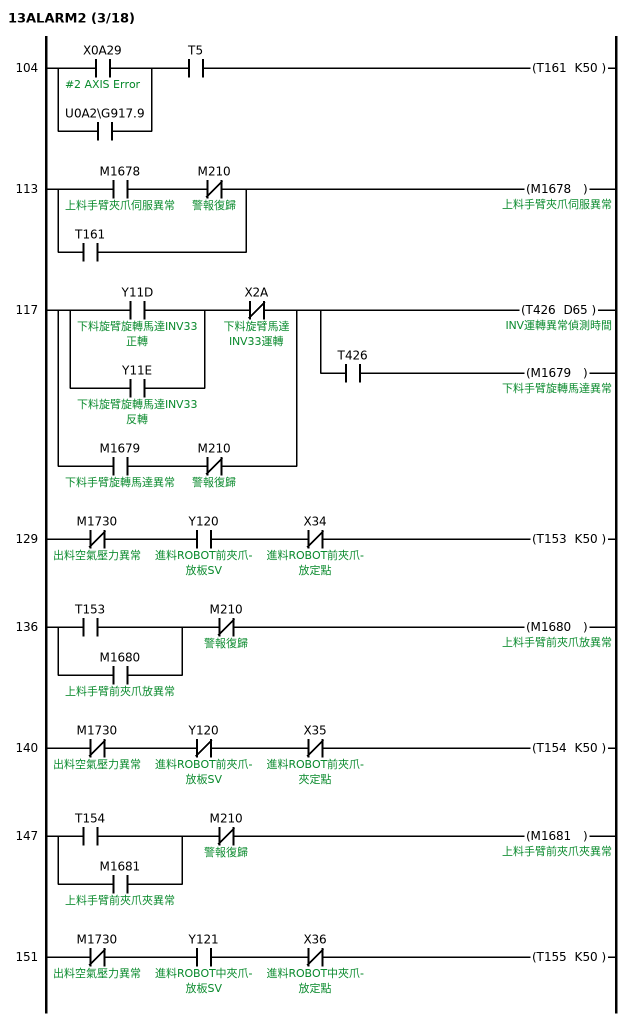
[picture p72: ladder of 13ALARM2, rungs at steps 104 to 151]
104   LD      X0A29  ; #2 AXIS Error
      OR      U0A2\G917.9
      AND     T5
      OUT     T161 K50
113   LD      M1678  ; 上料手臂夾爪伺服異常
      ANI     M210  ; 警報復歸
      OR      T161
      OUT     M1678  ; 上料手臂夾爪伺服異常
117   LD      Y11D  ; 下料旋臂旋轉馬達INV33正轉
      OR      Y11E  ; 下料旋臂旋轉馬達INV33反轉
      ANI     X2A  ; 下料旋臂馬達    INV33運轉
      LD      M1679  ; 下料手臂旋轉馬達異常
      ANI     M210  ; 警報復歸
      ORB
      OUT     T426 D65  ; INV運轉異常偵測時間
      AND     T426
      OUT     M1679  ; 下料手臂旋轉馬達異常
129   LDI     M1730  ; 出料空氣壓力異常
      AND     Y120  ; 進料ROBOT前夾爪-放板SV
      ANI     X34  ; 進料ROBOT前夾爪-放定點
      OUT     T153 K50
136   LD      T153
      OR      M1680  ; 上料手臂前夾爪放異常
      ANI     M210  ; 警報復歸
      OUT     M1680  ; 上料手臂前夾爪放異常
140   LDI     M1730  ; 出料空氣壓力異常
      ANI     Y120  ; 進料ROBOT前夾爪-放板SV
      ANI     X35  ; 進料ROBOT前夾爪-夾定點
      OUT     T154 K50
147   LD      T154
      OR      M1681  ; 上料手臂前夾爪夾異常
      ANI     M210  ; 警報復歸
      OUT     M1681  ; 上料手臂前夾爪夾異常
151   LDI     M1730  ; 出料空氣壓力異常
      AND     Y121  ; 進料ROBOT中夾爪-放板SV
      ANI     X36  ; 進料ROBOT中夾爪-放定點
      OUT     T155 K50
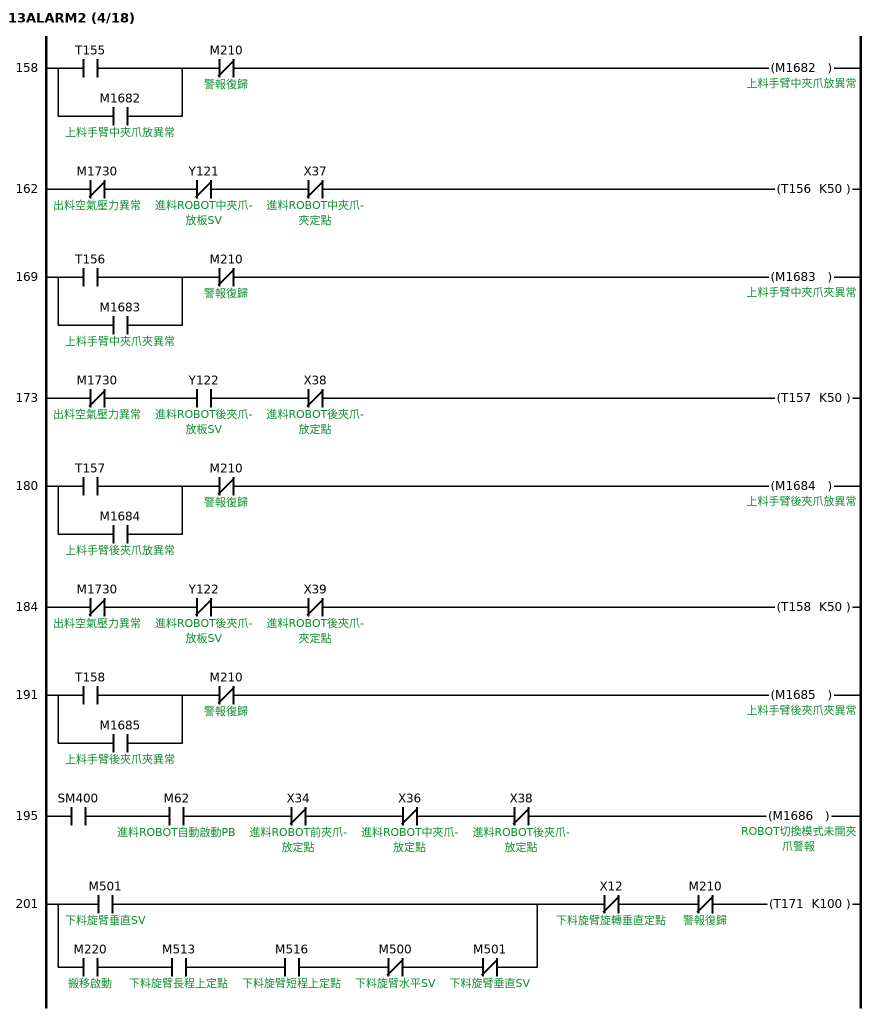
158   LD      T155
      OR      M1682  ; 上料手臂中夾爪放異常
      ANI     M210  ; 警報復歸
      OUT     M1682  ; 上料手臂中夾爪放異常
162   LDI     M1730  ; 出料空氣壓力異常
      ANI     Y121  ; 進料ROBOT中夾爪-放板SV
      ANI     X37  ; 進料ROBOT中夾爪-夾定點
      OUT     T156 K50
169   LD      T156
      OR      M1683  ; 上料手臂中夾爪夾異常
      ANI     M210  ; 警報復歸
      OUT     M1683  ; 上料手臂中夾爪夾異常
173   LDI     M1730  ; 出料空氣壓力異常
      AND     Y122  ; 進料ROBOT後夾爪-放板SV
      ANI     X38  ; 進料ROBOT後夾爪-放定點
      OUT     T157 K50
180   LD      T157
      OR      M1684  ; 上料手臂後夾爪放異常
      ANI     M210  ; 警報復歸
      OUT     M1684  ; 上料手臂後夾爪放異常
184   LDI     M1730  ; 出料空氣壓力異常
      ANI     Y122  ; 進料ROBOT後夾爪-放板SV
      ANI     X39  ; 進料ROBOT後夾爪-夾定點
      OUT     T158 K50
191   LD      T158
      OR      M1685  ; 上料手臂後夾爪夾異常
      ANI     M210  ; 警報復歸
      OUT     M1685  ; 上料手臂後夾爪夾異常
195   LD      SM400
      AND     M62  ; 進料ROBOT自動啟動PB
      ANI     X34  ; 進料ROBOT前夾爪-放定點
      ANI     X36  ; 進料ROBOT中夾爪-放定點
      ANI     X38  ; 進料ROBOT後夾爪-放定點
      OUT     M1686  ; ROBOT切換模式未開夾爪警報
201   LD      M501  ; 下料旋臂垂直SV
      LD      M220  ; 搬移啟動
      AND     M513  ; 下料旋臂長程上定點
      AND     M516  ; 下料旋臂短程上定點
      ANI     M500  ; 下料旋臂水平SV
      ANI     M501  ; 下料旋臂垂直SV
      ORB
      ANI     X12  ; 下料旋臂旋轉垂直定點
      ANI     M210  ; 警報復歸
      OUT     T171 K100
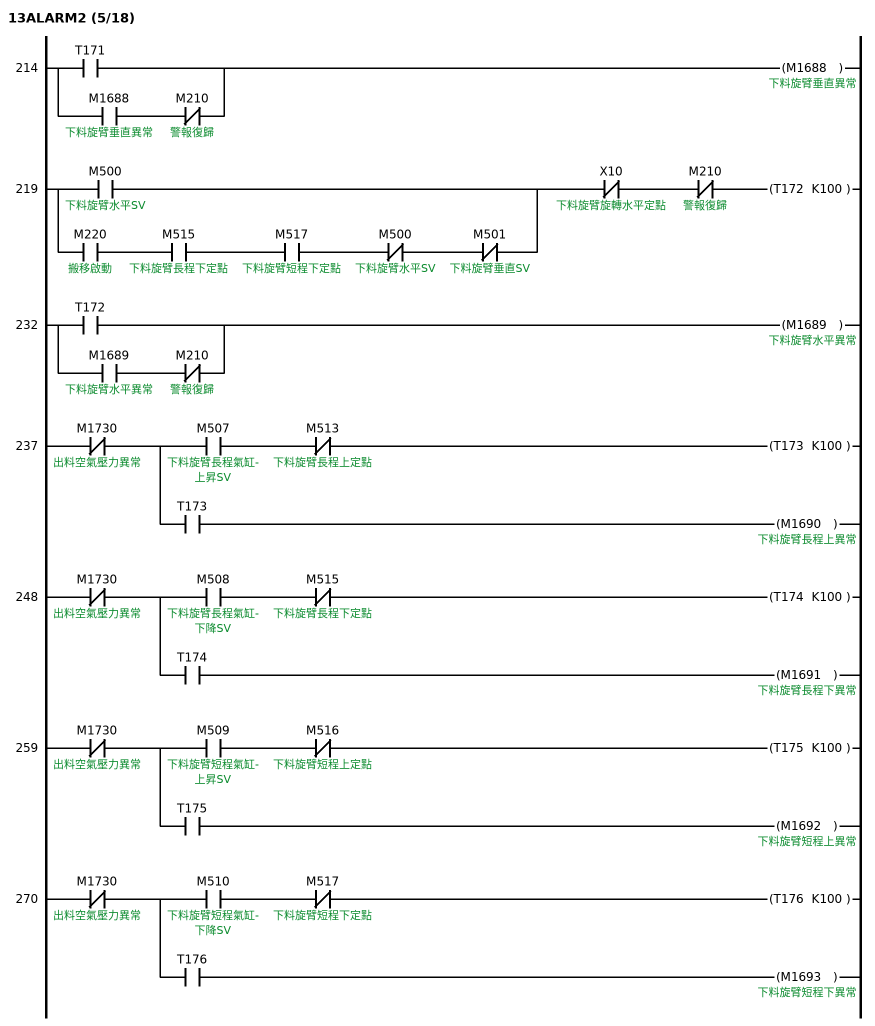
214   LD      T171
      LD      M1688  ; 下料旋臂垂直異常
      ANI     M210  ; 警報復歸
      ORB
      OUT     M1688  ; 下料旋臂垂直異常
219   LD      M500  ; 下料旋臂水平SV
      LD      M220  ; 搬移啟動
      AND     M515  ; 下料旋臂長程下定點
      AND     M517  ; 下料旋臂短程下定點
      ANI     M500  ; 下料旋臂水平SV
      ANI     M501  ; 下料旋臂垂直SV
      ORB
      ANI     X10  ; 下料旋臂旋轉水平定點
      ANI     M210  ; 警報復歸
      OUT     T172 K100
232   LD      T172
      LD      M1689  ; 下料旋臂水平異常
      ANI     M210  ; 警報復歸
      ORB
      OUT     M1689  ; 下料旋臂水平異常
237   LDI     M1730  ; 出料空氣壓力異常
      MPS
      AND     M507  ; 下料旋臂長程氣缸-上昇SV
      ANI     M513  ; 下料旋臂長程上定點
      OUT     T173 K100
      MPP
      AND     T173
      OUT     M1690  ; 下料旋臂長程上異常
248   LDI     M1730  ; 出料空氣壓力異常
      MPS
      AND     M508  ; 下料旋臂長程氣缸-下降SV
      ANI     M515  ; 下料旋臂長程下定點
      OUT     T174 K100
      MPP
      AND     T174
      OUT     M1691  ; 下料旋臂長程下異常
259   LDI     M1730  ; 出料空氣壓力異常
      MPS
      AND     M509  ; 下料旋臂短程氣缸-上昇SV
      ANI     M516  ; 下料旋臂短程上定點
      OUT     T175 K100
      MPP
      AND     T175
      OUT     M1692  ; 下料旋臂短程上異常
270   LDI     M1730  ; 出料空氣壓力異常
      MPS
      AND     M510  ; 下料旋臂短程氣缸-下降SV
      ANI     M517  ; 下料旋臂短程下定點
      OUT     T176 K100
      MPP
      AND     T176
      OUT     M1693  ; 下料旋臂短程下異常
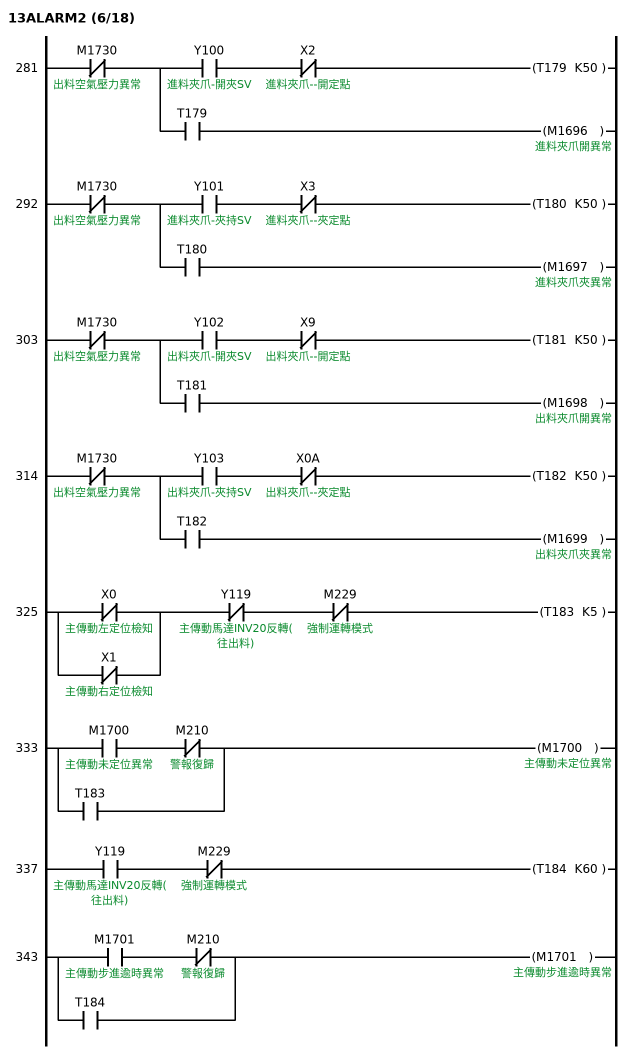
281   LDI     M1730  ; 出料空氣壓力異常
      MPS
      AND     Y100  ; 進料夾爪-開夾SV
      ANI     X2  ; 進料夾爪--開定點
      OUT     T179 K50
      MPP
      AND     T179
      OUT     M1696  ; 進料夾爪開異常
292   LDI     M1730  ; 出料空氣壓力異常
      MPS
      AND     Y101  ; 進料夾爪-夾持SV
      ANI     X3  ; 進料夾爪--夾定點
      OUT     T180 K50
      MPP
      AND     T180
      OUT     M1697  ; 進料夾爪夾異常
303   LDI     M1730  ; 出料空氣壓力異常
      MPS
      AND     Y102  ; 出料夾爪-開夾SV
      ANI     X9  ; 出料夾爪--開定點
      OUT     T181 K50
      MPP
      AND     T181
      OUT     M1698  ; 出料夾爪開異常
314   LDI     M1730  ; 出料空氣壓力異常
      MPS
      AND     Y103  ; 出料夾爪-夾持SV
      ANI     X0A  ; 出料夾爪--夾定點
      OUT     T182 K50
      MPP
      AND     T182
      OUT     M1699  ; 出料夾爪夾異常
325   LDI     X0  ; 主傳動左定位檢知
      ORI     X1  ; 主傳動右定位檢知
      ANI     Y119  ; 主傳動馬達INV20反轉(往出料)
      ANI     M229  ; 強制運轉模式
      OUT     T183 K5
333   LD      M1700  ; 主傳動未定位異常
      ANI     M210  ; 警報復歸
      OR      T183
      OUT     M1700  ; 主傳動未定位異常
337   LD      Y119  ; 主傳動馬達INV20反轉(往出料)
      ANI     M229  ; 強制運轉模式
      OUT     T184 K60
343   LD      M1701  ; 主傳動步進逾時異常
      ANI     M210  ; 警報復歸
      OR      T184
      OUT     M1701  ; 主傳動步進逾時異常
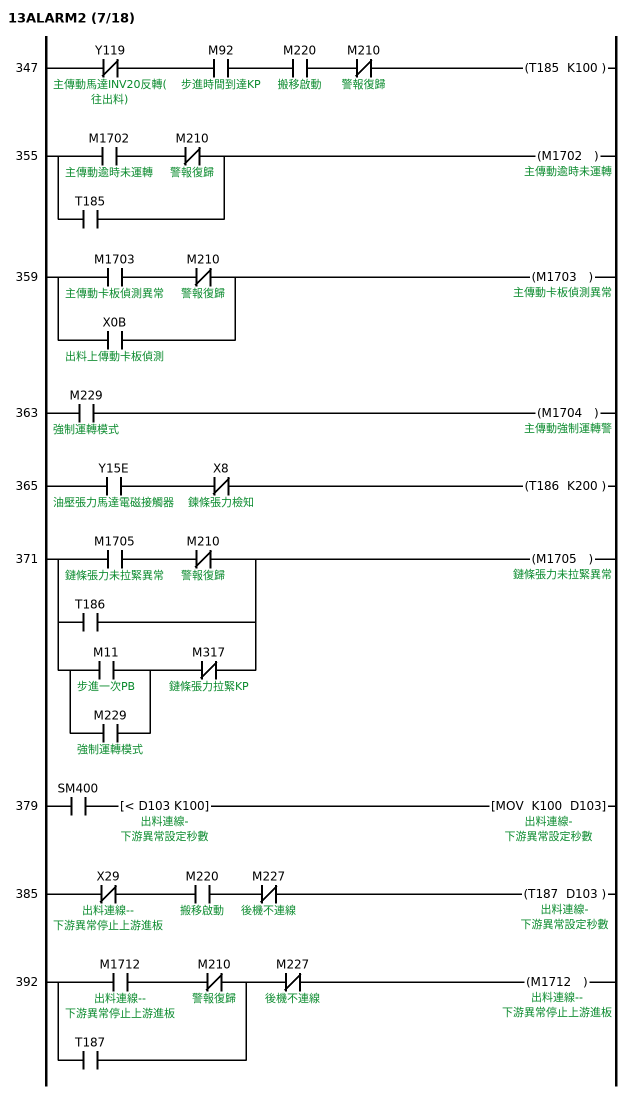
347   LDI     Y119  ; 主傳動馬達INV20反轉(往出料)
      AND     M92  ; 步進時間到達KP
      AND     M220  ; 搬移啟動
      ANI     M210  ; 警報復歸
      OUT     T185 K100
355   LD      M1702  ; 主傳動逾時未運轉
      ANI     M210  ; 警報復歸
      OR      T185
      OUT     M1702  ; 主傳動逾時未運轉
359   LD      M1703  ; 主傳動卡板偵測異常
      ANI     M210  ; 警報復歸
      OR      X0B  ; 出料上傳動卡板偵測
      OUT     M1703  ; 主傳動卡板偵測異常
363   LD      M229  ; 強制運轉模式
      OUT     M1704  ; 主傳動強制運轉警
365   LD      Y15E  ; 油壓張力馬達電磁接觸器
      ANI     X8  ; 鍊條張力檢知
      OUT     T186 K200
371   LD      M1705  ; 鏈條張力未拉緊異常
      ANI     M210  ; 警報復歸
      OR      T186
      LD      M11  ; 步進一次PB
      OR      M229  ; 強制運轉模式
      ANI     M317  ; 鏈條張力拉緊KP
      ORB
      OUT     M1705  ; 鏈條張力未拉緊異常
379   LD      SM400
      AND<    D103 K100  ; 出料連線-下游異常設定秒數
      MOV     K100 D103
385   LDI     X29  ; 出料連線--下游異常停止上游進板
      AND     M220  ; 搬移啟動
      ANI     M227  ; 後機不連線
      OUT     T187 D103  ; 出料連線-下游異常設定秒數
392   LD      M1712  ; 出料連線--下游異常停止上游進板
      ANI     M210  ; 警報復歸
      OR      T187
      ANI     M227  ; 後機不連線
      OUT     M1712  ; 出料連線--下游異常停止上游進板
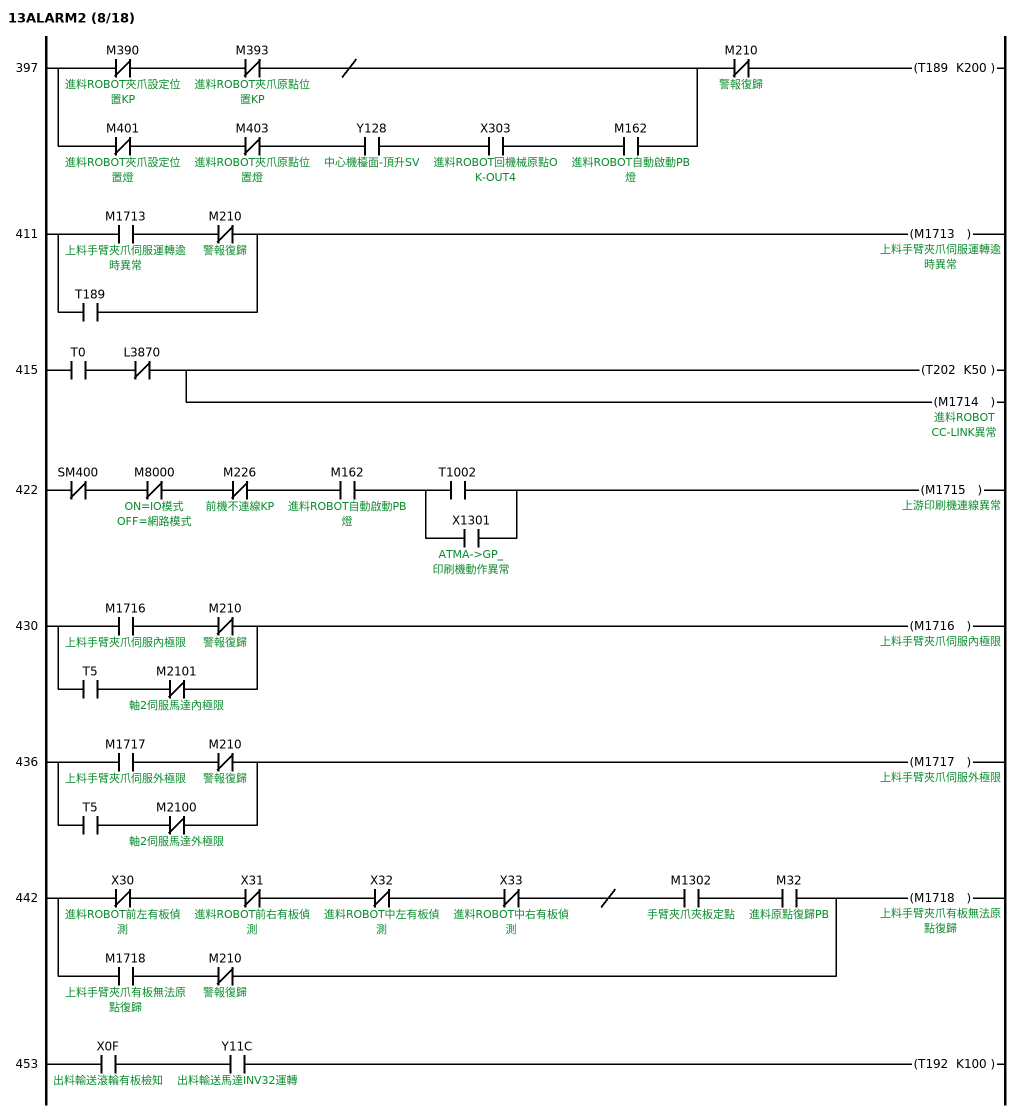
397   LDI     M390  ; 進料ROBOT夾爪設定位置KP
      ANI     M393  ; 進料ROBOT夾爪原點位置KP
      INV
      LDI     M401  ; 進料ROBOT夾爪設定位置燈
      ANI     M403  ; 進料ROBOT夾爪原點位置燈
      AND     Y128  ; 中心機檯面-頂升SV
      AND     X303  ; 進料ROBOT回機械原點OK-OUT4
      AND     M162  ; 進料ROBOT自動啟動PB燈
      ORB
      ANI     M210  ; 警報復歸
      OUT     T189 K200
411   LD      M1713  ; 上料手臂夾爪伺服運轉逾時異常
      ANI     M210  ; 警報復歸
      OR      T189
      OUT     M1713  ; 上料手臂夾爪伺服運轉逾時異常
415   LD      T0
      ANI     L3870
      OUT     T202 K50
      OUT     M1714  ; 進料ROBOT CC-LINK異常
422   LDI     SM400
      ANI     M8000  ; ON=IO模式 OFF=網路模式
      ANI     M226  ; 前機不連線KP
      AND     M162  ; 進料ROBOT自動啟動PB燈
      LD      T1002
      OR      X1301  ; ATMA->GP_印刷機動作異常
      ANB
      OUT     M1715  ; 上游印刷機連線異常
430   LD      M1716  ; 上料手臂夾爪伺服內極限
      ANI     M210  ; 警報復歸
      LD      T5
      ANI     M2101  ; 軸2伺服馬達內極限
      ORB
      OUT     M1716  ; 上料手臂夾爪伺服內極限
436   LD      M1717  ; 上料手臂夾爪伺服外極限
      ANI     M210  ; 警報復歸
      LD      T5
      ANI     M2100  ; 軸2伺服馬達外極限
      ORB
      OUT     M1717  ; 上料手臂夾爪伺服外極限
442   LDI     X30  ; 進料ROBOT前左有板偵測
      ANI     X31  ; 進料ROBOT前右有板偵測
      ANI     X32  ; 進料ROBOT中左有板偵測
      ANI     X33  ; 進料ROBOT中右有板偵測
      INV
      AND     M1302  ; 手臂夾爪夾板定點
      AND     M32  ; 進料原點復歸PB
      LD      M1718  ; 上料手臂夾爪有板無法原點復歸
      ANI     M210  ; 警報復歸
      ORB
      OUT     M1718  ; 上料手臂夾爪有板無法原點復歸
453   LD      X0F  ; 出料輸送滾輪有板檢知
      AND     Y11C  ; 出料輸送馬達INV32運轉
      OUT     T192 K100
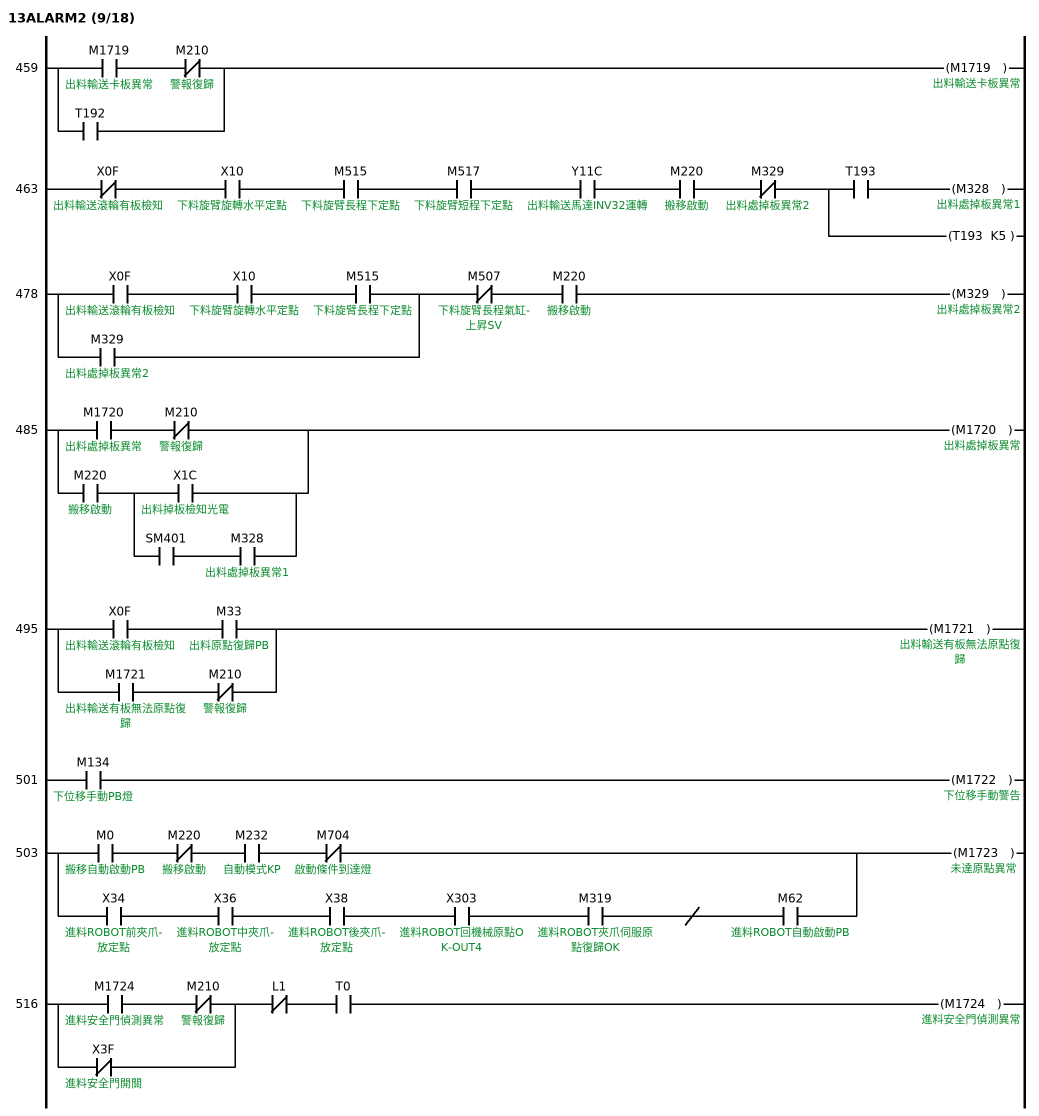
459   LD      M1719  ; 出料輸送卡板異常
      ANI     M210  ; 警報復歸
      OR      T192
      OUT     M1719  ; 出料輸送卡板異常
463   LDI     X0F  ; 出料輸送滾輪有板檢知
      AND     X10  ; 下料旋臂旋轉水平定點
      AND     M515  ; 下料旋臂長程下定點
      AND     M517  ; 下料旋臂短程下定點
      AND     Y11C  ; 出料輸送馬達INV32運轉
      AND     M220  ; 搬移啟動
      ANI     M329  ; 出料處掉板異常2
      MPS
      AND     T193
      OUT     M328  ; 出料處掉板異常1
      MPP
      OUT     T193 K5
478   LD      X0F  ; 出料輸送滾輪有板檢知
      AND     X10  ; 下料旋臂旋轉水平定點
      AND     M515  ; 下料旋臂長程下定點
      OR      M329  ; 出料處掉板異常2
      ANI     M507  ; 下料旋臂長程氣缸-上昇SV
      AND     M220  ; 搬移啟動
      OUT     M329  ; 出料處掉板異常2
485   LD      M1720  ; 出料處掉板異常
      ANI     M210  ; 警報復歸
      LD      M220  ; 搬移啟動
      LD      X1C  ; 出料掉板檢知光電
      LD      SM401
      AND     M328  ; 出料處掉板異常1
      ORB
      ANB
      ORB
      OUT     M1720  ; 出料處掉板異常
495   LD      X0F  ; 出料輸送滾輪有板檢知
      AND     M33  ; 出料原點復歸PB
      LD      M1721  ; 出料輸送有板無法原點復歸
      ANI     M210  ; 警報復歸
      ORB
      OUT     M1721  ; 出料輸送有板無法原點復歸
501   LD      M134  ; 下位移手動PB燈
      OUT     M1722  ; 下位移手動警告
503   LD      M0  ; 搬移自動啟動PB
      ANI     M220  ; 搬移啟動
      AND     M232  ; 自動模式KP
      ANI     M704  ; 啟動條件到達燈
      LD      X34  ; 進料ROBOT前夾爪-放定點
      AND     X36  ; 進料ROBOT中夾爪-放定點
      AND     X38  ; 進料ROBOT後夾爪-放定點
      AND     X303  ; 進料ROBOT回機械原點OK-OUT4
      AND     M319  ; 進料ROBOT夾爪伺服原點復歸OK
      INV
      AND     M62  ; 進料ROBOT自動啟動PB
      ORB
      OUT     M1723  ; 未達原點異常
516   LD      M1724  ; 進料安全門偵測異常
      ANI     M210  ; 警報復歸
      ORI     X3F  ; 進料安全門開關
      ANI     L1
      AND     T0
      OUT     M1724  ; 進料安全門偵測異常
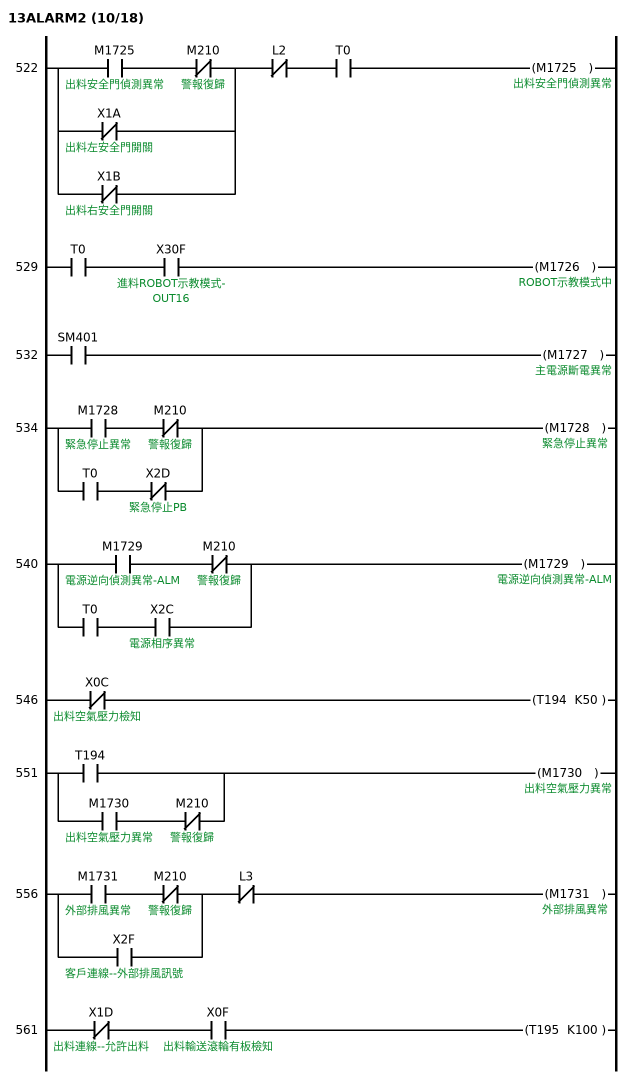
522   LD      M1725  ; 出料安全門偵測異常
      ANI     M210  ; 警報復歸
      ORI     X1A  ; 出料左安全門開關
      ORI     X1B  ; 出料右安全門開關
      ANI     L2
      AND     T0
      OUT     M1725  ; 出料安全門偵測異常
529   LD      T0
      AND     X30F  ; 進料ROBOT示教模式-OUT16
      OUT     M1726  ; ROBOT示教模式中
532   LD      SM401
      OUT     M1727  ; 主電源斷電異常
534   LD      M1728  ; 緊急停止異常
      ANI     M210  ; 警報復歸
      LD      T0
      ANI     X2D  ; 緊急停止PB
      ORB
      OUT     M1728  ; 緊急停止異常
540   LD      M1729  ; 電源逆向偵測異常-ALM
      ANI     M210  ; 警報復歸
      LD      T0
      AND     X2C  ; 電源相序異常
      ORB
      OUT     M1729  ; 電源逆向偵測異常-ALM
546   LDI     X0C  ; 出料空氣壓力檢知
      OUT     T194 K50
551   LD      T194
      LD      M1730  ; 出料空氣壓力異常
      ANI     M210  ; 警報復歸
      ORB
      OUT     M1730  ; 出料空氣壓力異常
556   LD      M1731  ; 外部排風異常
      ANI     M210  ; 警報復歸
      OR      X2F  ; 客戶連線--外部排風訊號
      ANI     L3
      OUT     M1731  ; 外部排風異常
561   LDI     X1D  ; 出料連線--允許出料
      AND     X0F  ; 出料輸送滾輪有板檢知
      OUT     T195 K100
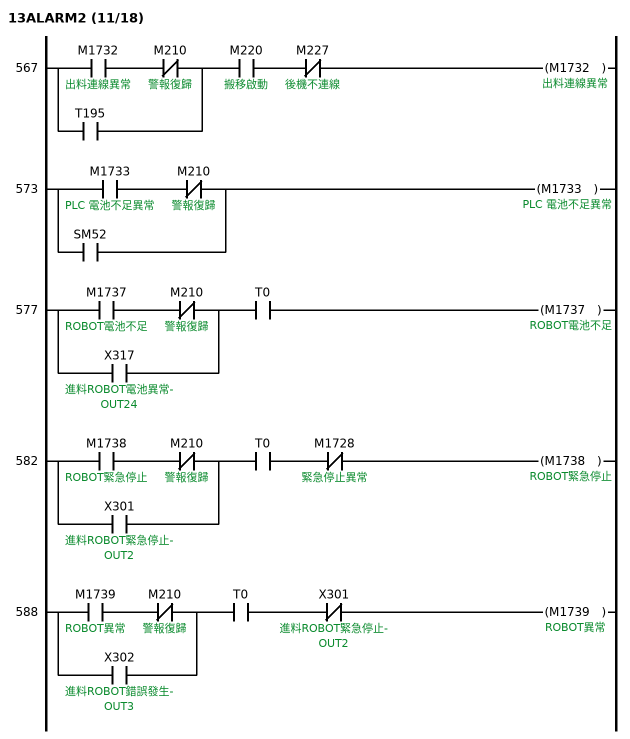
567   LD      M1732  ; 出料連線異常
      ANI     M210  ; 警報復歸
      OR      T195
      AND     M220  ; 搬移啟動
      ANI     M227  ; 後機不連線
      OUT     M1732  ; 出料連線異常
573   LD      M1733  ; PLC 電池不足異常
      ANI     M210  ; 警報復歸
      OR      SM52
      OUT     M1733  ; PLC 電池不足異常
577   LD      M1737  ; ROBOT電池不足
      ANI     M210  ; 警報復歸
      OR      X317  ; 進料ROBOT電池異常-OUT24
      AND     T0
      OUT     M1737  ; ROBOT電池不足
582   LD      M1738  ; ROBOT緊急停止
      ANI     M210  ; 警報復歸
      OR      X301  ; 進料ROBOT緊急停止-OUT2
      AND     T0
      ANI     M1728  ; 緊急停止異常
      OUT     M1738  ; ROBOT緊急停止
588   LD      M1739  ; ROBOT異常
      ANI     M210  ; 警報復歸
      OR      X302  ; 進料ROBOT錯誤發生-OUT3
      AND     T0
      ANI     X301  ; 進料ROBOT緊急停止-OUT2
      OUT     M1739  ; ROBOT異常
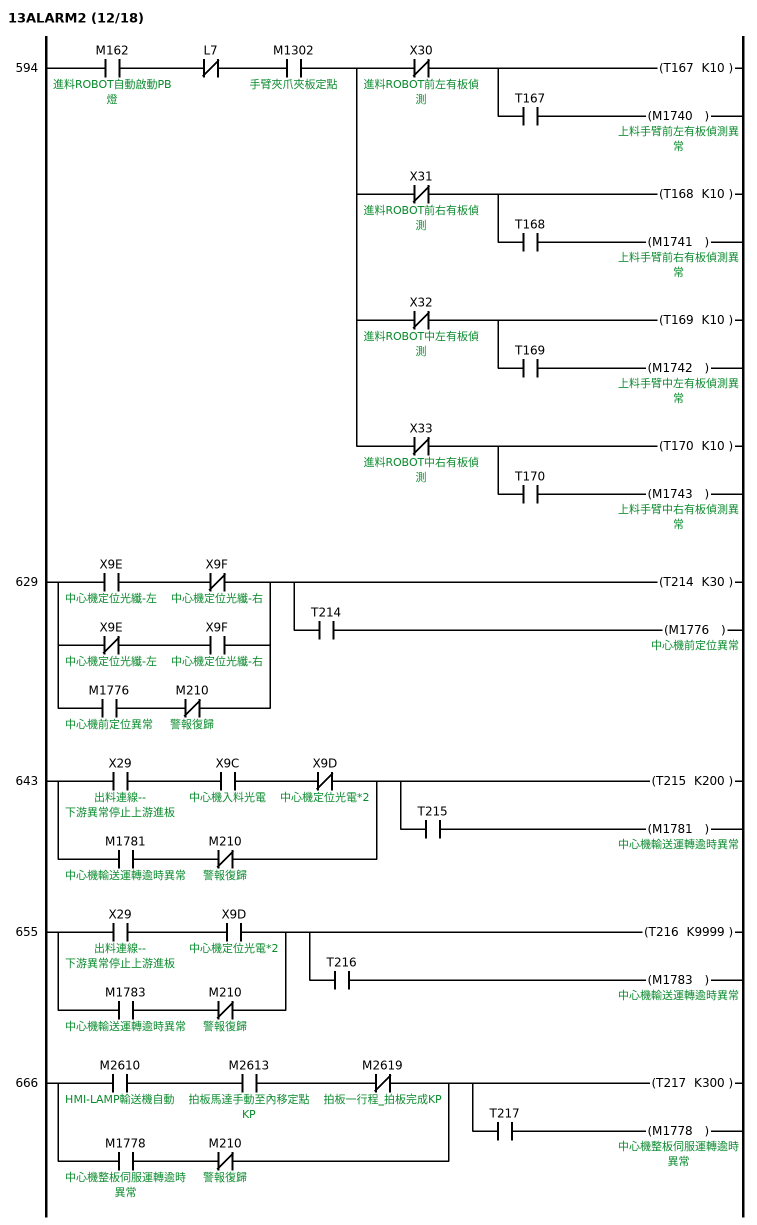
594   LD      M162  ; 進料ROBOT自動啟動PB燈
      ANI     L7
      AND     M1302  ; 手臂夾爪夾板定點
      MPS
      ANI     X30  ; 進料ROBOT前左有板偵測
      OUT     T167 K10
      AND     T167
      OUT     M1740  ; 上料手臂前左有板偵測異常
      MRD
      ANI     X31  ; 進料ROBOT前右有板偵測
      OUT     T168 K10
      AND     T168
      OUT     M1741  ; 上料手臂前右有板偵測異常
      MRD
      ANI     X32  ; 進料ROBOT中左有板偵測
      OUT     T169 K10
      AND     T169
      OUT     M1742  ; 上料手臂中左有板偵測異常
      MPP
      ANI     X33  ; 進料ROBOT中右有板偵測
      OUT     T170 K10
      AND     T170
      OUT     M1743  ; 上料手臂中右有板偵測異常
629   LD      X9E  ; 中心機定位光纖-左
      ANI     X9F  ; 中心機定位光纖-右
      LDI     X9E  ; 中心機定位光纖-左
      AND     X9F  ; 中心機定位光纖-右
      ORB
      LD      M1776  ; 中心機前定位異常
      ANI     M210  ; 警報復歸
      ORB
      OUT     T214 K30
      AND     T214
      OUT     M1776  ; 中心機前定位異常
643   LD      X29  ; 出料連線--下游異常停止上游進板
      AND     X9C  ; 中心機入料光電
      ANI     X9D  ; 中心機定位光電*2
      LD      M1781  ; 中心機輸送運轉逾時異常
      ANI     M210  ; 警報復歸
      ORB
      OUT     T215 K200
      AND     T215
      OUT     M1781  ; 中心機輸送運轉逾時異常
655   LD      X29  ; 出料連線--下游異常停止上游進板
      AND     X9D  ; 中心機定位光電*2
      LD      M1783  ; 中心機輸送運轉逾時異常
      ANI     M210  ; 警報復歸
      ORB
      OUT     T216 K9999
      AND     T216
      OUT     M1783  ; 中心機輸送運轉逾時異常
666   LD      M2610  ; HMI-LAMP輸送機自動
      AND     M2613  ; 拍板馬達手動至內移定點KP
      ANI     M2619  ; 拍板一行程_拍板完成KP
      LD      M1778  ; 中心機整板伺服運轉逾時異常
      ANI     M210  ; 警報復歸
      ORB
      OUT     T217 K300
      AND     T217
      OUT     M1778  ; 中心機整板伺服運轉逾時異常
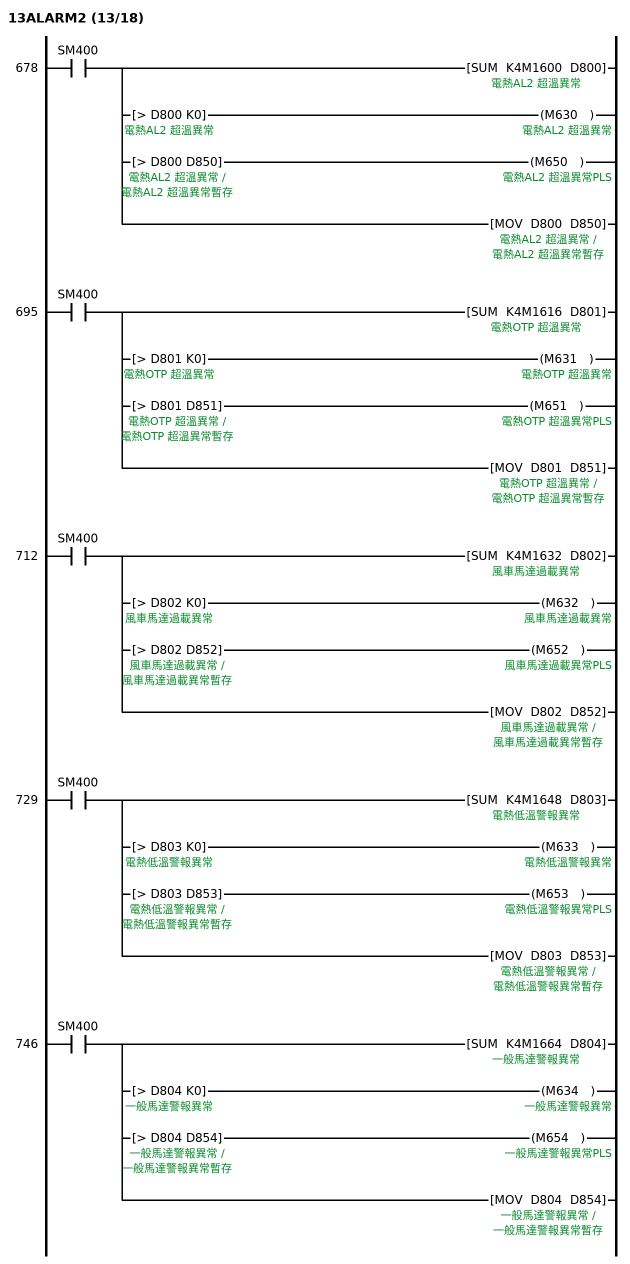
678   LD      SM400
      SUM     K4M1600 D800  ; #01 電熱AL2 超溫 / 電熱AL2 超溫異常
      MPS
      AND>    D800 K0  ; 電熱AL2 超溫異常
      OUT     M630  ; 電熱AL2 超溫異常
      MRD
      AND>    D800 D850  ; 電熱AL2 超溫異常 / 電熱AL2 超溫異常暫存
      OUT     M650  ; 電熱AL2 超溫異常PLS
      MPP
      MOV     D800 D850
695   LD      SM400
      SUM     K4M1616 D801  ; #01 電熱OTP 超溫 / 電熱OTP 超溫異常
      MPS
      AND>    D801 K0  ; 電熱OTP 超溫異常
      OUT     M631  ; 電熱OTP 超溫異常
      MRD
      AND>    D801 D851  ; 電熱OTP 超溫異常 / 電熱OTP 超溫異常暫存
      OUT     M651  ; 電熱OTP 超溫異常PLS
      MPP
      MOV     D801 D851
712   LD      SM400
      SUM     K4M1632 D802  ; #01 風車過載 / 風車馬達過載異常
      MPS
      AND>    D802 K0  ; 風車馬達過載異常
      OUT     M632  ; 風車馬達過載異常
      MRD
      AND>    D802 D852  ; 風車馬達過載異常 / 風車馬達過載異常暫存
      OUT     M652  ; 風車馬達過載異常PLS
      MPP
      MOV     D802 D852
729   LD      SM400
      SUM     K4M1648 D803  ; #01 低溫警報 / 電熱低溫警報異常
      MPS
      AND>    D803 K0  ; 電熱低溫警報異常
      OUT     M633  ; 電熱低溫警報異常
      MRD
      AND>    D803 D853  ; 電熱低溫警報異常 / 電熱低溫警報異常暫存
      OUT     M653  ; 電熱低溫警報異常PLS
      MPP
      MOV     D803 D853
746   LD      SM400
      SUM     K4M1664 D804  ; 一般馬達警報異常
      MPS
      AND>    D804 K0  ; 一般馬達警報異常
      OUT     M634  ; 一般馬達警報異常
      MRD
      AND>    D804 D854  ; 一般馬達警報異常 / 一般馬達警報異常暫存
      OUT     M654  ; 一般馬達警報異常PLS
      MPP
      MOV     D804 D854
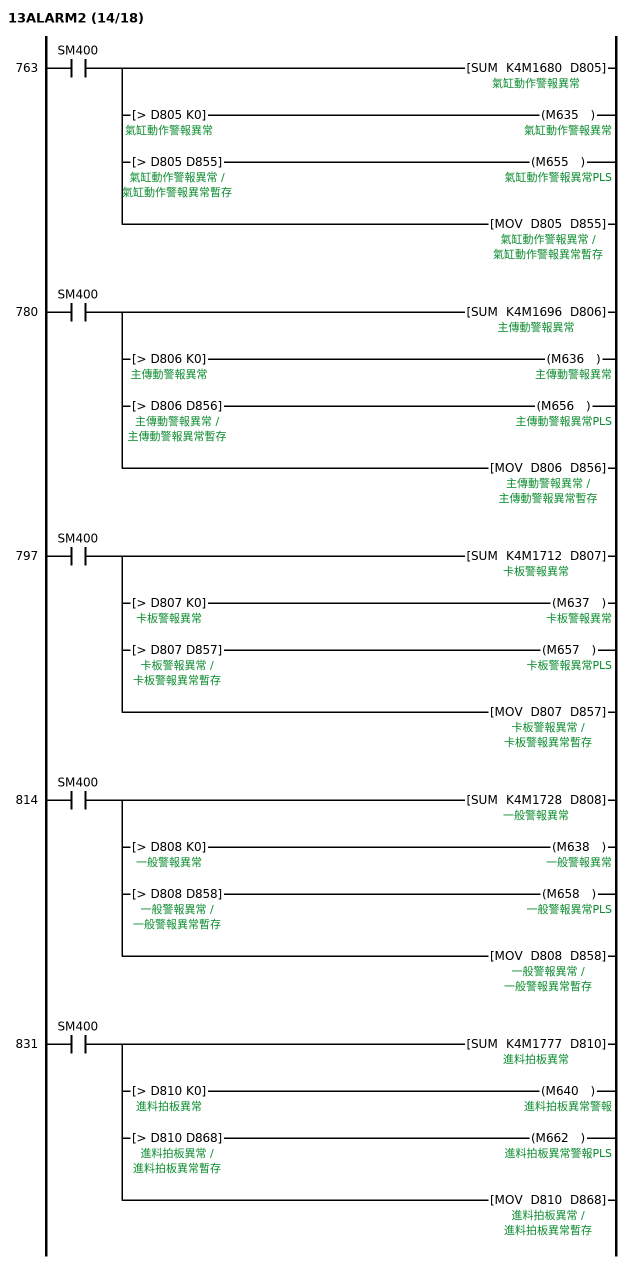
763   LD      SM400
      SUM     K4M1680 D805  ; 氣缸動作警報異常
      MPS
      AND>    D805 K0  ; 氣缸動作警報異常
      OUT     M635  ; 氣缸動作警報異常
      MRD
      AND>    D805 D855  ; 氣缸動作警報異常 / 氣缸動作警報異常暫存
      OUT     M655  ; 氣缸動作警報異常PLS
      MPP
      MOV     D805 D855
780   LD      SM400
      SUM     K4M1696 D806  ; 主傳動警報異常
      MPS
      AND>    D806 K0  ; 主傳動警報異常
      OUT     M636  ; 主傳動警報異常
      MRD
      AND>    D806 D856  ; 主傳動警報異常 / 主傳動警報異常暫存
      OUT     M656  ; 主傳動警報異常PLS
      MPP
      MOV     D806 D856
797   LD      SM400
      SUM     K4M1712 D807  ; 卡板警報異常
      MPS
      AND>    D807 K0  ; 卡板警報異常
      OUT     M637  ; 卡板警報異常
      MRD
      AND>    D807 D857  ; 卡板警報異常 / 卡板警報異常暫存
      OUT     M657  ; 卡板警報異常PLS
      MPP
      MOV     D807 D857
814   LD      SM400
      SUM     K4M1728 D808  ; 一般警報異常
      MPS
      AND>    D808 K0  ; 一般警報異常
      OUT     M638  ; 一般警報異常
      MRD
      AND>    D808 D858  ; 一般警報異常 / 一般警報異常暫存
      OUT     M658  ; 一般警報異常PLS
      MPP
      MOV     D808 D858
831   LD      SM400
      SUM     K4M1777 D810  ; 輸送機輸送變頻器異常-ALM / 進料拍板異常
      MPS
      AND>    D810 K0  ; 進料拍板異常
      OUT     M640  ; 進料拍板異常警報
      MRD
      AND>    D810 D868  ; 進料拍板異常 / 進料拍板異常暫存
      OUT     M662  ; 進料拍板異常警報PLS
      MPP
      MOV     D810 D868
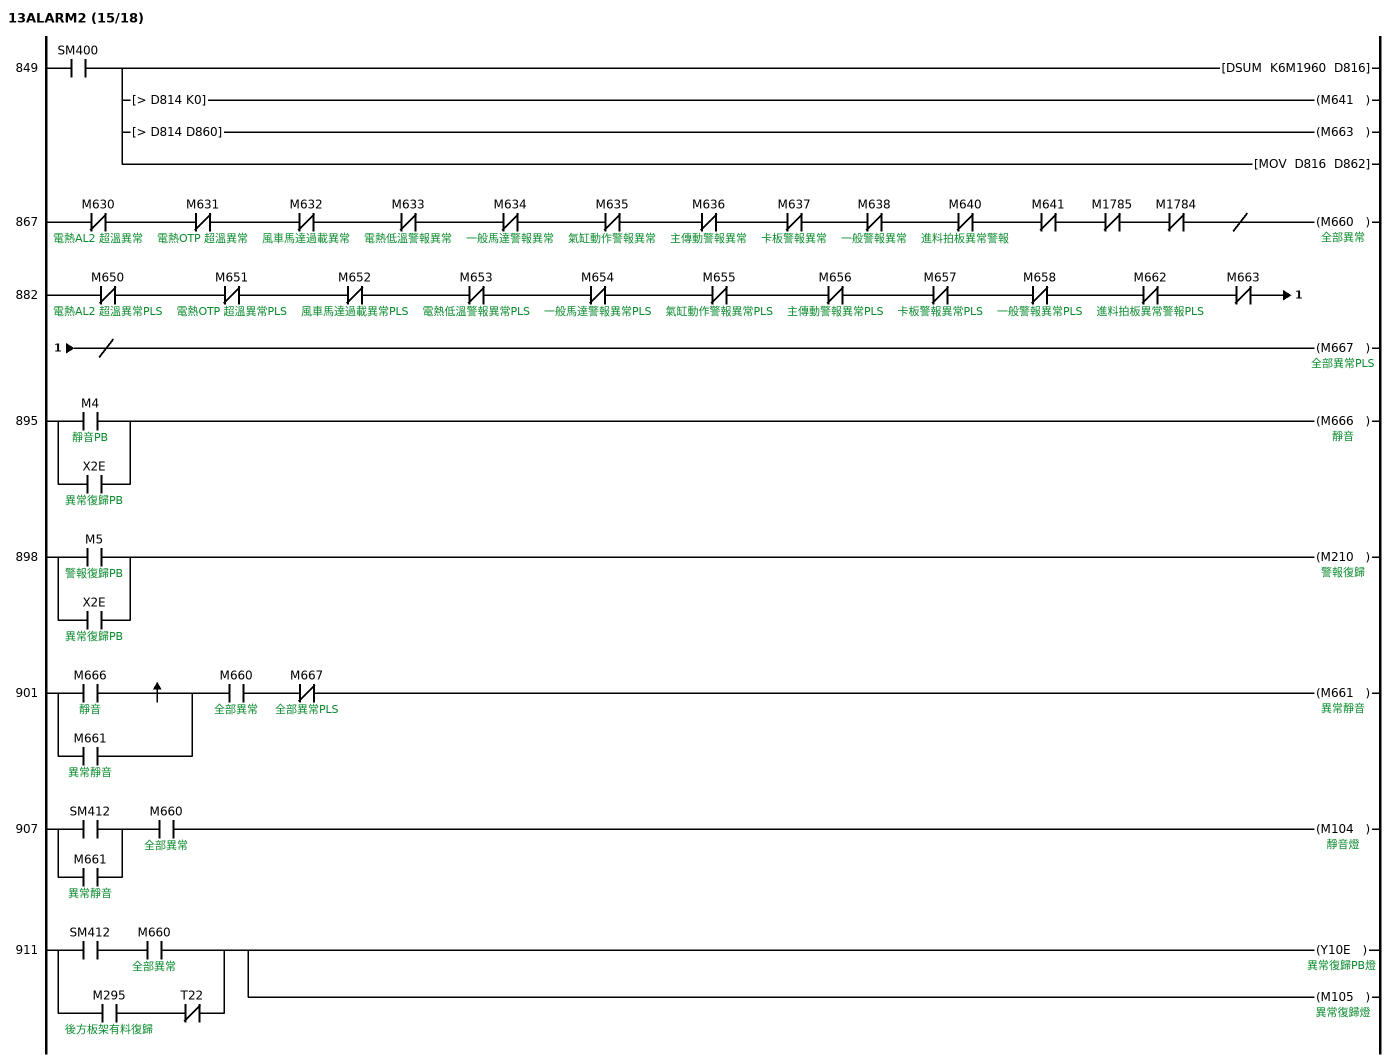
849   LD      SM400
      DSUM    K6M1960 D816
      MPS
      AND>    D814 K0
      OUT     M641
      MRD
      AND>    D814 D860
      OUT     M663
      MPP
      MOV     D816 D862
867   LDI     M630  ; 電熱AL2 超溫異常
      ANI     M631  ; 電熱OTP 超溫異常
      ANI     M632  ; 風車馬達過載異常
      ANI     M633  ; 電熱低溫警報異常
      ANI     M634  ; 一般馬達警報異常
      ANI     M635  ; 氣缸動作警報異常
      ANI     M636  ; 主傳動警報異常
      ANI     M637  ; 卡板警報異常
      ANI     M638  ; 一般警報異常
      ANI     M640  ; 進料拍板異常警報
      ANI     M641
      ANI     M1785
      ANI     M1784
      INV
      OUT     M660  ; 全部異常
882   LDI     M650  ; 電熱AL2 超溫異常PLS
      ANI     M651  ; 電熱OTP 超溫異常PLS
      ANI     M652  ; 風車馬達過載異常PLS
      ANI     M653  ; 電熱低溫警報異常PLS
      ANI     M654  ; 一般馬達警報異常PLS
      ANI     M655  ; 氣缸動作警報異常PLS
      ANI     M656  ; 主傳動警報異常PLS
      ANI     M657  ; 卡板警報異常PLS
      ANI     M658  ; 一般警報異常PLS
      ANI     M662  ; 進料拍板異常警報PLS
      ANI     M663
      INV
      OUT     M667  ; 全部異常PLS
895   LD      M4  ; 靜音PB
      OR      X2E  ; 異常復歸PB
      OUT     M666  ; 靜音
898   LD      M5  ; 警報復歸PB
      OR      X2E  ; 異常復歸PB
      OUT     M210  ; 警報復歸
901   LD      M666  ; 靜音
      MEP
      OR      M661  ; 異常靜音
      AND     M660  ; 全部異常
      ANI     M667  ; 全部異常PLS
      OUT     M661  ; 異常靜音
907   LD      SM412
      OR      M661  ; 異常靜音
      AND     M660  ; 全部異常
      OUT     M104  ; 靜音燈
911   LD      SM412
      AND     M660  ; 全部異常
      LD      M295  ; 後方板架有料復歸
      ANI     T22
      ORB
      OUT     Y10E  ; 異常復歸PB燈
      OUT     M105  ; 異常復歸燈
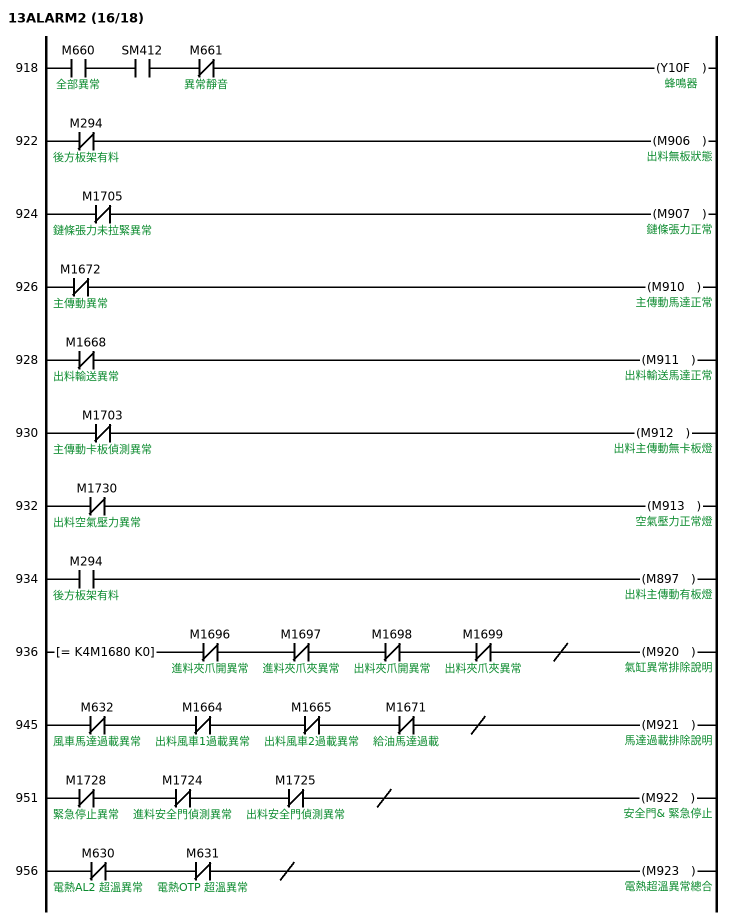
918   LD      M660  ; 全部異常
      AND     SM412
      ANI     M661  ; 異常靜音
      OUT     Y10F  ; 蜂鳴器
922   LDI     M294  ; 後方板架有料
      OUT     M906  ; 出料無板狀態
924   LDI     M1705  ; 鏈條張力未拉緊異常
      OUT     M907  ; 鏈條張力正常
926   LDI     M1672  ; 主傳動異常
      OUT     M910  ; 主傳動馬達正常
928   LDI     M1668  ; 出料輸送異常
      OUT     M911  ; 出料輸送馬達正常
930   LDI     M1703  ; 主傳動卡板偵測異常
      OUT     M912  ; 出料主傳動無卡板燈
932   LDI     M1730  ; 出料空氣壓力異常
      OUT     M913  ; 空氣壓力正常燈
934   LD      M294  ; 後方板架有料
      OUT     M897  ; 出料主傳動有板燈
936   LD=     K4M1680 K0  ; 上料手臂前夾爪放異常
      ANI     M1696  ; 進料夾爪開異常
      ANI     M1697  ; 進料夾爪夾異常
      ANI     M1698  ; 出料夾爪開異常
      ANI     M1699  ; 出料夾爪夾異常
      INV
      OUT     M920  ; 氣缸異常排除說明
945   LDI     M632  ; 風車馬達過載異常
      ANI     M1664  ; 出料風車1過載異常
      ANI     M1665  ; 出料風車2過載異常
      ANI     M1671  ; 給油馬達過載
      INV
      OUT     M921  ; 馬達過載排除說明
951   LDI     M1728  ; 緊急停止異常
      ANI     M1724  ; 進料安全門偵測異常
      ANI     M1725  ; 出料安全門偵測異常
      INV
      OUT     M922  ; 安全門& 緊急停止
956   LDI     M630  ; 電熱AL2 超溫異常
      ANI     M631  ; 電熱OTP 超溫異常
      INV
      OUT     M923  ; 電熱超溫異常總合
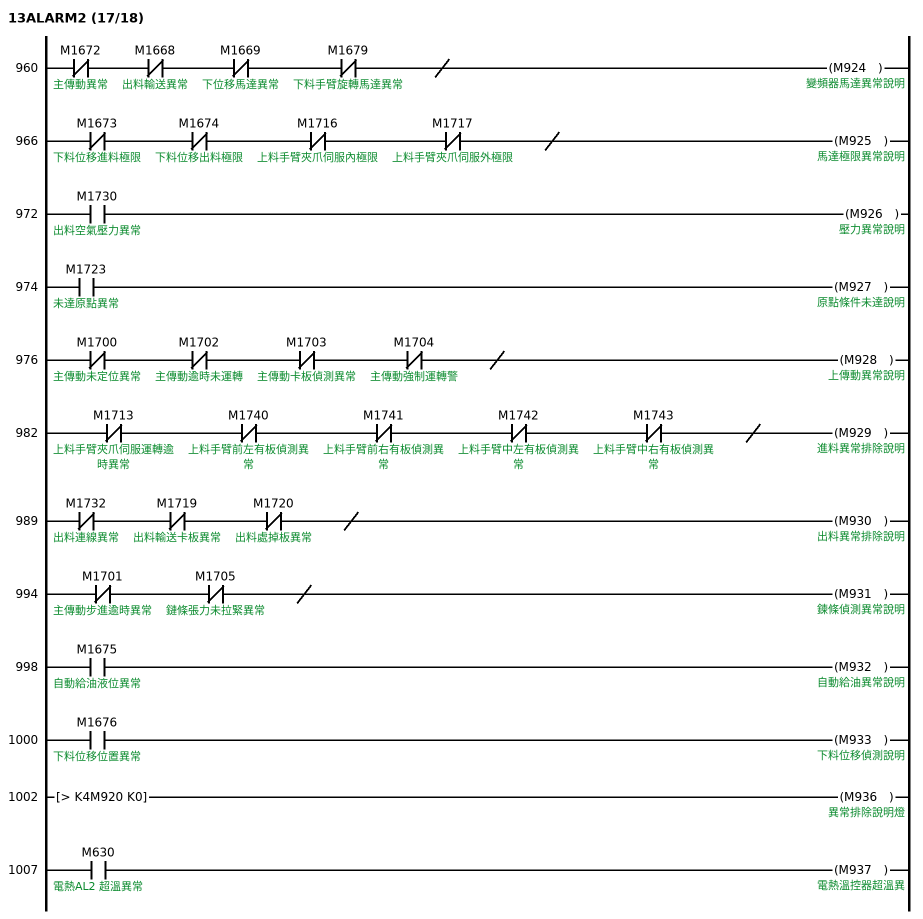
960   LDI     M1672  ; 主傳動異常
      ANI     M1668  ; 出料輸送異常
      ANI     M1669  ; 下位移馬達異常
      ANI     M1679  ; 下料手臂旋轉馬達異常
      INV
      OUT     M924  ; 變頻器馬達異常說明
966   LDI     M1673  ; 下料位移進料極限
      ANI     M1674  ; 下料位移出料極限
      ANI     M1716  ; 上料手臂夾爪伺服內極限
      ANI     M1717  ; 上料手臂夾爪伺服外極限
      INV
      OUT     M925  ; 馬達極限異常說明
972   LD      M1730  ; 出料空氣壓力異常
      OUT     M926  ; 壓力異常說明
974   LD      M1723  ; 未達原點異常
      OUT     M927  ; 原點條件未達說明
976   LDI     M1700  ; 主傳動未定位異常
      ANI     M1702  ; 主傳動逾時未運轉
      ANI     M1703  ; 主傳動卡板偵測異常
      ANI     M1704  ; 主傳動強制運轉警
      INV
      OUT     M928  ; 上傳動異常說明
982   LDI     M1713  ; 上料手臂夾爪伺服運轉逾時異常
      ANI     M1740  ; 上料手臂前左有板偵測異常
      ANI     M1741  ; 上料手臂前右有板偵測異常
      ANI     M1742  ; 上料手臂中左有板偵測異常
      ANI     M1743  ; 上料手臂中右有板偵測異常
      INV
      OUT     M929  ; 進料異常排除說明
989   LDI     M1732  ; 出料連線異常
      ANI     M1719  ; 出料輸送卡板異常
      ANI     M1720  ; 出料處掉板異常
      INV
      OUT     M930  ; 出料異常排除說明
994   LDI     M1701  ; 主傳動步進逾時異常
      ANI     M1705  ; 鏈條張力未拉緊異常
      INV
      OUT     M931  ; 鍊條偵測異常說明
998   LD      M1675  ; 自動給油液位異常
      OUT     M932  ; 自動給油異常說明
1000  LD      M1676  ; 下料位移位置異常
      OUT     M933  ; 下料位移偵測說明
1002  LD>     K4M920 K0  ; 氣缸異常排除說明
      OUT     M936  ; 異常排除說明燈
1007  LD      M630  ; 電熱AL2 超溫異常
      OUT     M937  ; 電熱溫控器超溫異
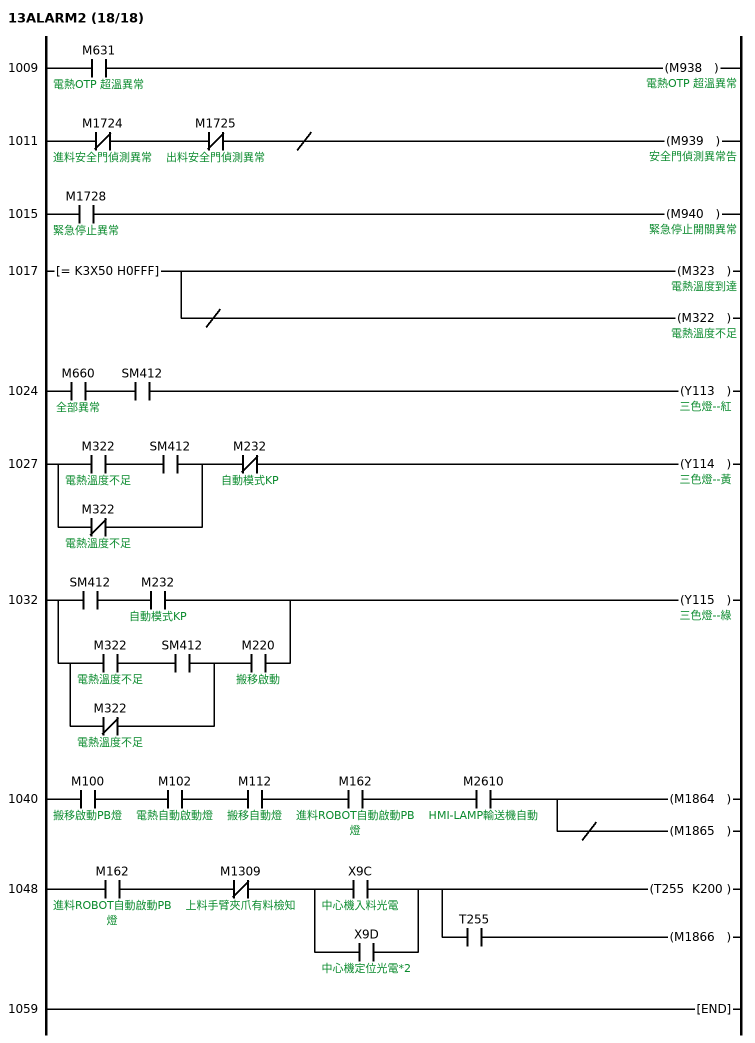
1009  LD      M631  ; 電熱OTP 超溫異常
      OUT     M938  ; 電熱OTP 超溫異常
1011  LDI     M1724  ; 進料安全門偵測異常
      ANI     M1725  ; 出料安全門偵測異常
      INV
      OUT     M939  ; 安全門偵測異常告
1015  LD      M1728  ; 緊急停止異常
      OUT     M940  ; 緊急停止開關異常
1017  LD=     K3X50 H0FFF  ; NO,01   溫度到達AL1
      OUT     M323  ; 電熱溫度到達
      INV
      OUT     M322  ; 電熱溫度不足
1024  LD      M660  ; 全部異常
      AND     SM412
      OUT     Y113  ; 三色燈--紅
1027  LD      M322  ; 電熱溫度不足
      AND     SM412
      ORI     M322  ; 電熱溫度不足
      ANI     M232  ; 自動模式KP
      OUT     Y114  ; 三色燈--黃
1032  LD      SM412
      AND     M232  ; 自動模式KP
      LD      M322  ; 電熱溫度不足
      AND     SM412
      ORI     M322  ; 電熱溫度不足
      AND     M220  ; 搬移啟動
      ORB
      OUT     Y115  ; 三色燈--綠
1040  LD      M100  ; 搬移啟動PB燈
      AND     M102  ; 電熱自動啟動燈
      AND     M112  ; 搬移自動燈
      AND     M162  ; 進料ROBOT自動啟動PB燈
      AND     M2610  ; HMI-LAMP輸送機自動
      OUT     M1864
      INV
      OUT     M1865
1048  LD      M162  ; 進料ROBOT自動啟動PB燈
      ANI     M1309  ; 上料手臂夾爪有料檢知
      LD      X9C  ; 中心機入料光電
      OR      X9D  ; 中心機定位光電*2
      ANB
      OUT     T255 K200
      AND     T255
      OUT     M1866
1059  END
END_PROGRAM

PROGRAM 14TIME
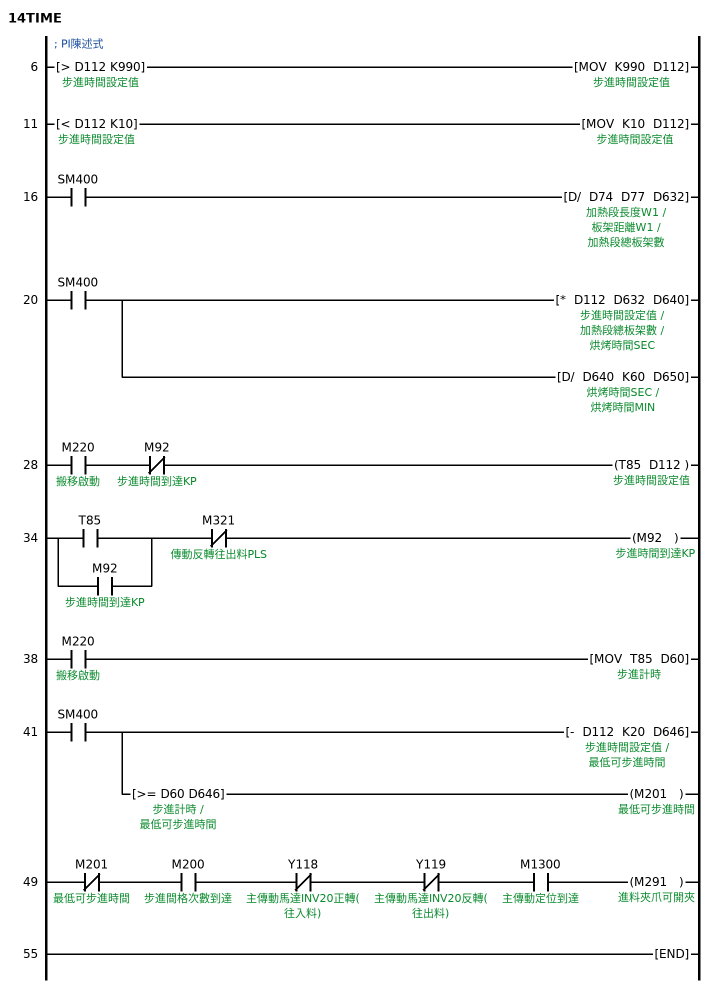
; PI陳述式
6     LD>     D112 K990  ; 步進時間設定值
      MOV     K990 D112
11    LD<     D112 K10  ; 步進時間設定值
      MOV     K10 D112
16    LD      SM400
      D/      D74 D77 D632  ; 加熱段長度W1 / 板架距離W1 / 加熱段總板架數
20    LD      SM400
      *       D112 D632 D640  ; 烘烤時間SEC
      D/      D640 K60 D650  ; 烘烤時間MIN
28    LD      M220  ; 搬移啟動
      ANI     M92  ; 步進時間到達KP
      OUT     T85 D112  ; 步進時間設定值
34    LD      T85
      OR      M92  ; 步進時間到達KP
      ANI     M321  ; 傳動反轉往出料PLS
      OUT     M92  ; 步進時間到達KP
38    LD      M220  ; 搬移啟動
      MOV     T85 D60  ; 步進計時
41    LD      SM400
      -       D112 K20 D646  ; 最低可步進時間
      AND>=   D60 D646  ; 步進計時 / 最低可步進時間
      OUT     M201  ; 最低可步進時間
49    LDI     M201  ; 最低可步進時間
      AND     M200  ; 步進間格次數到達
      ANI     Y118  ; 主傳動馬達INV20正轉(往入料)
      ANI     Y119  ; 主傳動馬達INV20反轉(往出料)
      AND     M1300  ; 主傳動定位到達
      OUT     M291  ; 進料夾爪可開夾
55    END
END_PROGRAM

PROGRAM 15STATUS
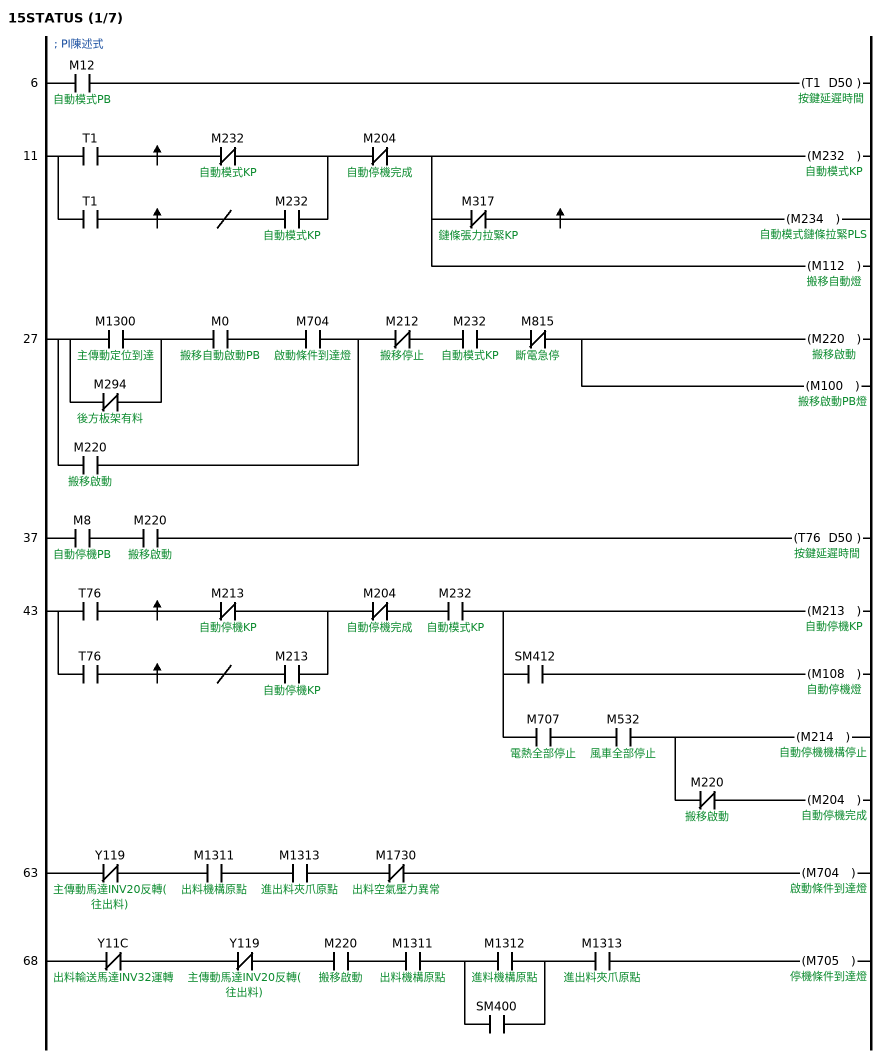
; PI陳述式
6     LD      M12  ; 自動模式PB
      OUT     T1 D50  ; 按鍵延遲時間
11    LD      T1
      MEP
      ANI     M232  ; 自動模式KP
      LD      T1
      MEP
      INV
      AND     M232  ; 自動模式KP
      ORB
      ANI     M204  ; 自動停機完成
      OUT     M232  ; 自動模式KP
      MPS
      ANI     M317  ; 鏈條張力拉緊KP
      MEP
      OUT     M234  ; 自動模式鏈條拉緊PLS
      MPP
      OUT     M112  ; 搬移自動燈
27    LD      M1300  ; 主傳動定位到達
      ORI     M294  ; 後方板架有料
      AND     M0  ; 搬移自動啟動PB
      AND     M704  ; 啟動條件到達燈
      OR      M220  ; 搬移啟動
      ANI     M212  ; 搬移停止
      AND     M232  ; 自動模式KP
      ANI     M815  ; 斷電急停
      OUT     M220  ; 搬移啟動
      OUT     M100  ; 搬移啟動PB燈
37    LD      M8  ; 自動停機PB
      AND     M220  ; 搬移啟動
      OUT     T76 D50  ; 按鍵延遲時間
43    LD      T76
      MEP
      ANI     M213  ; 自動停機KP
      LD      T76
      MEP
      INV
      AND     M213  ; 自動停機KP
      ORB
      ANI     M204  ; 自動停機完成
      AND     M232  ; 自動模式KP
      OUT     M213  ; 自動停機KP
      MPS
      AND     SM412
      OUT     M108  ; 自動停機燈
      MPP
      AND     M707  ; 電熱全部停止
      AND     M532  ; 風車全部停止
      OUT     M214  ; 自動停機機構停止
      ANI     M220  ; 搬移啟動
      OUT     M204  ; 自動停機完成
63    LDI     Y119  ; 主傳動馬達INV20反轉(往出料)
      AND     M1311  ; 出料機構原點
      AND     M1313  ; 進出料夾爪原點
      ANI     M1730  ; 出料空氣壓力異常
      OUT     M704  ; 啟動條件到達燈
68    LDI     Y11C  ; 出料輸送馬達INV32運轉
      ANI     Y119  ; 主傳動馬達INV20反轉(往出料)
      AND     M220  ; 搬移啟動
      AND     M1311  ; 出料機構原點
      LD      M1312  ; 進料機構原點
      OR      SM400
      ANB
      AND     M1313  ; 進出料夾爪原點
      OUT     M705  ; 停機條件到達燈
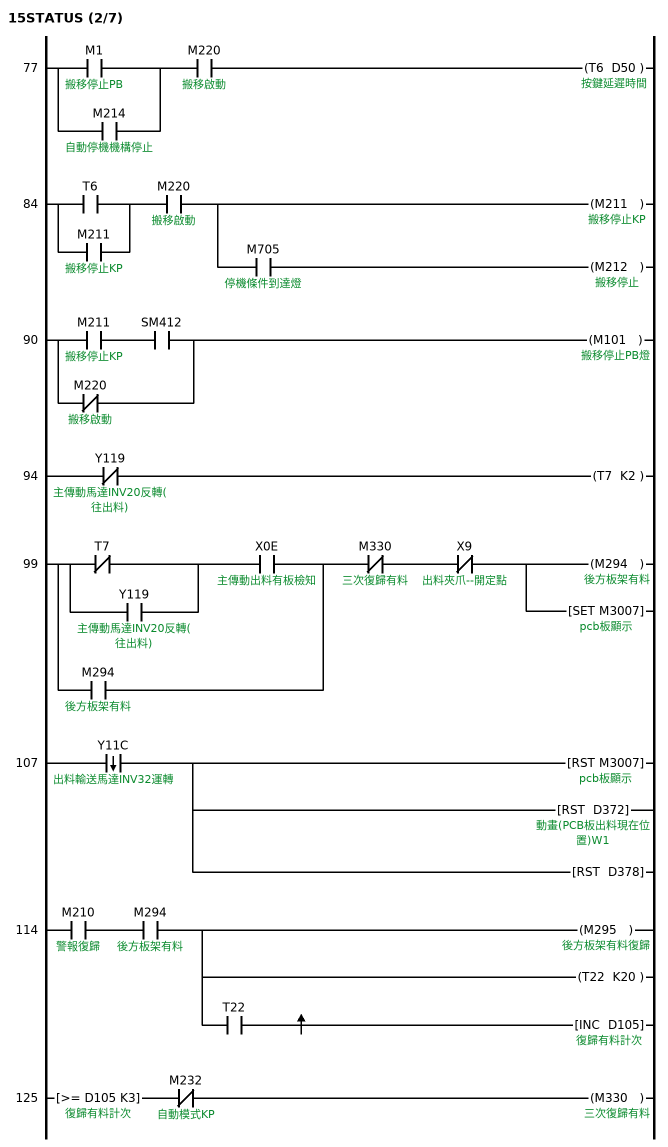
77    LD      M1  ; 搬移停止PB
      OR      M214  ; 自動停機機構停止
      AND     M220  ; 搬移啟動
      OUT     T6 D50  ; 按鍵延遲時間
84    LD      T6
      OR      M211  ; 搬移停止KP
      AND     M220  ; 搬移啟動
      OUT     M211  ; 搬移停止KP
      AND     M705  ; 停機條件到達燈
      OUT     M212  ; 搬移停止
90    LD      M211  ; 搬移停止KP
      AND     SM412
      ORI     M220  ; 搬移啟動
      OUT     M101  ; 搬移停止PB燈
94    LDI     Y119  ; 主傳動馬達INV20反轉(往出料)
      OUT     T7 K2
99    LDI     T7
      OR      Y119  ; 主傳動馬達INV20反轉(往出料)
      AND     X0E  ; 主傳動出料有板檢知
      OR      M294  ; 後方板架有料
      ANI     M330  ; 三次復歸有料
      ANI     X9  ; 出料夾爪--開定點
      OUT     M294  ; 後方板架有料
      SET     M3007  ; pcb板顯示
107   LDF     Y11C  ; 出料輸送馬達INV32運轉
      RST     M3007  ; pcb板顯示
      RST     D372  ; 動畫(PCB板出料現在位置)W1
      RST     D378
114   LD      M210  ; 警報復歸
      AND     M294  ; 後方板架有料
      OUT     M295  ; 後方板架有料復歸
      OUT     T22 K20
      AND     T22
      MEP
      INC     D105  ; 復歸有料計次
125   LD>=    D105 K3  ; 復歸有料計次
      ANI     M232  ; 自動模式KP
      OUT     M330  ; 三次復歸有料
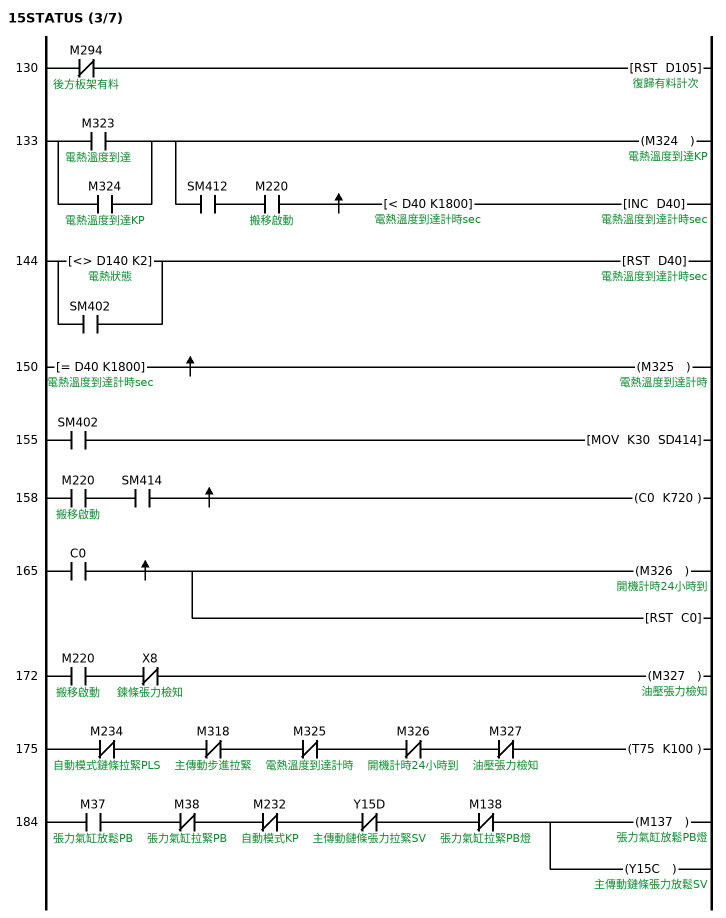
130   LDI     M294  ; 後方板架有料
      RST     D105  ; 復歸有料計次
133   LD      M323  ; 電熱溫度到達
      OR      M324  ; 電熱溫度到達KP
      OUT     M324  ; 電熱溫度到達KP
      AND     SM412
      AND     M220  ; 搬移啟動
      MEP
      AND<    D40 K1800  ; 電熱溫度到達計時sec
      INC     D40
144   LD<>    D140 K2  ; 電熱狀態
      OR      SM402
      RST     D40  ; 電熱溫度到達計時sec
150   LD=     D40 K1800  ; 電熱溫度到達計時sec
      MEP
      OUT     M325  ; 電熱溫度到達計時
155   LD      SM402
      MOV     K30 SD414
158   LD      M220  ; 搬移啟動
      AND     SM414
      MEP
      OUT     C0 K720
165   LD      C0
      MEP
      OUT     M326  ; 開機計時24小時到
      RST     C0
172   LD      M220  ; 搬移啟動
      ANI     X8  ; 鍊條張力檢知
      OUT     M327  ; 油壓張力檢知
175   LDI     M234  ; 自動模式鏈條拉緊PLS
      ANI     M318  ; 主傳動步進拉緊
      ANI     M325  ; 電熱溫度到達計時
      ANI     M326  ; 開機計時24小時到
      ANI     M327  ; 油壓張力檢知
      OUT     T75 K100
184   LD      M37  ; 張力氣缸放鬆PB
      ANI     M38  ; 張力氣缸拉緊PB
      ANI     M232  ; 自動模式KP
      ANI     Y15D  ; 主傳動鏈條張力拉緊SV
      ANI     M138  ; 張力氣缸拉緊PB燈
      OUT     M137  ; 張力氣缸放鬆PB燈
      OUT     Y15C  ; 主傳動鏈條張力放鬆SV
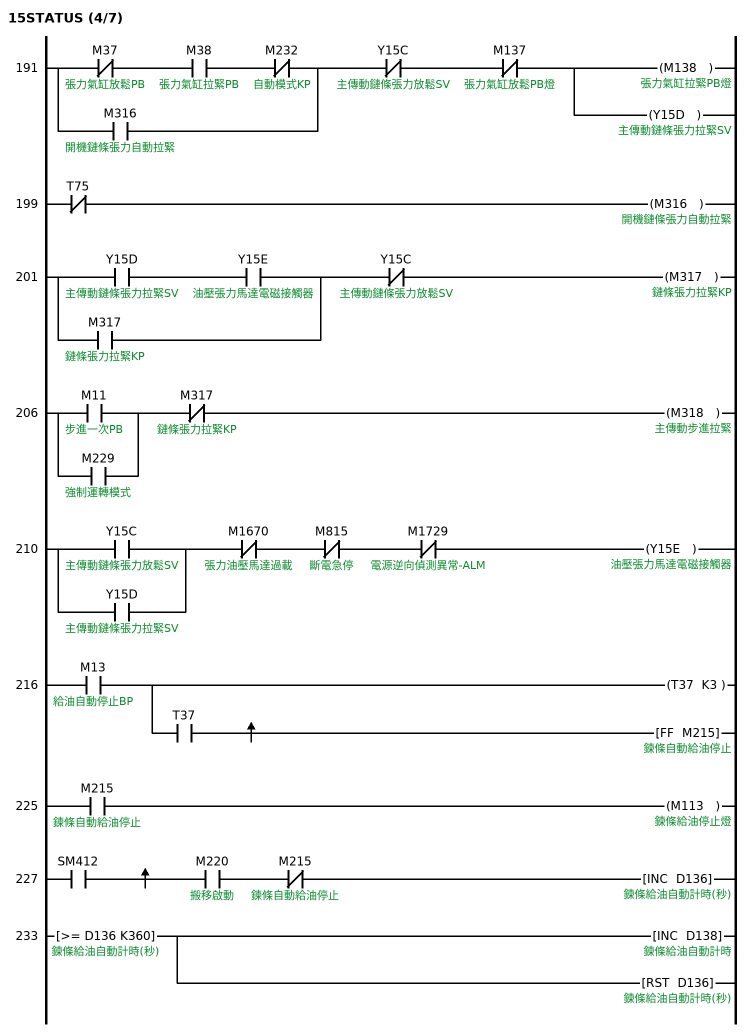
191   LDI     M37  ; 張力氣缸放鬆PB
      AND     M38  ; 張力氣缸拉緊PB
      ANI     M232  ; 自動模式KP
      OR      M316  ; 開機鏈條張力自動拉緊
      ANI     Y15C  ; 主傳動鏈條張力放鬆SV
      ANI     M137  ; 張力氣缸放鬆PB燈
      OUT     M138  ; 張力氣缸拉緊PB燈
      OUT     Y15D  ; 主傳動鏈條張力拉緊SV
199   LDI     T75
      OUT     M316  ; 開機鏈條張力自動拉緊
201   LD      Y15D  ; 主傳動鏈條張力拉緊SV
      AND     Y15E  ; 油壓張力馬達電磁接觸器
      OR      M317  ; 鏈條張力拉緊KP
      ANI     Y15C  ; 主傳動鏈條張力放鬆SV
      OUT     M317  ; 鏈條張力拉緊KP
206   LD      M11  ; 步進一次PB
      OR      M229  ; 強制運轉模式
      ANI     M317  ; 鏈條張力拉緊KP
      OUT     M318  ; 主傳動步進拉緊
210   LD      Y15C  ; 主傳動鏈條張力放鬆SV
      OR      Y15D  ; 主傳動鏈條張力拉緊SV
      ANI     M1670  ; 張力油壓馬達過載
      ANI     M815  ; 斷電急停
      ANI     M1729  ; 電源逆向偵測異常-ALM
      OUT     Y15E  ; 油壓張力馬達電磁接觸器
216   LD      M13  ; 給油自動停止BP
      OUT     T37 K3
      AND     T37
      MEP
      FF      M215  ; 鍊條自動給油停止
225   LD      M215  ; 鍊條自動給油停止
      OUT     M113  ; 鍊條給油停止燈
227   LD      SM412
      MEP
      AND     M220  ; 搬移啟動
      ANI     M215  ; 鍊條自動給油停止
      INC     D136  ; 鍊條給油自動計時(秒)
233   LD>=    D136 K360  ; 鍊條給油自動計時(秒)
      INC     D138  ; 鍊條給油自動計時
      RST     D136  ; 鍊條給油自動計時(秒)
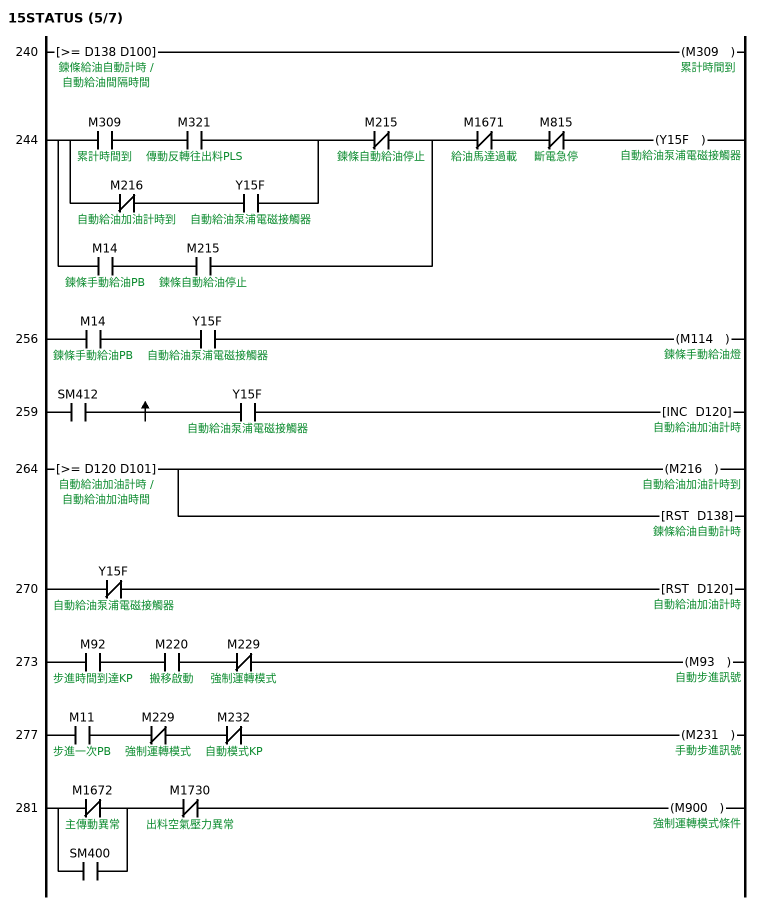
240   LD>=    D138 D100  ; 鍊條給油自動計時 / 自動給油間隔時間
      OUT     M309  ; 累計時間到
244   LD      M309  ; 累計時間到
      AND     M321  ; 傳動反轉往出料PLS
      LDI     M216  ; 自動給油加油計時到
      AND     Y15F  ; 自動給油泵浦電磁接觸器
      ORB
      ANI     M215  ; 鍊條自動給油停止
      LD      M14  ; 鍊條手動給油PB
      AND     M215  ; 鍊條自動給油停止
      ORB
      ANI     M1671  ; 給油馬達過載
      ANI     M815  ; 斷電急停
      OUT     Y15F  ; 自動給油泵浦電磁接觸器
256   LD      M14  ; 鍊條手動給油PB
      AND     Y15F  ; 自動給油泵浦電磁接觸器
      OUT     M114  ; 鍊條手動給油燈
259   LD      SM412
      MEP
      AND     Y15F  ; 自動給油泵浦電磁接觸器
      INC     D120  ; 自動給油加油計時
264   LD>=    D120 D101  ; 自動給油加油計時 / 自動給油加油時間
      OUT     M216  ; 自動給油加油計時到
      RST     D138  ; 鍊條給油自動計時
270   LDI     Y15F  ; 自動給油泵浦電磁接觸器
      RST     D120  ; 自動給油加油計時
273   LD      M92  ; 步進時間到達KP
      AND     M220  ; 搬移啟動
      ANI     M229  ; 強制運轉模式
      OUT     M93  ; 自動步進訊號
277   LD      M11  ; 步進一次PB
      ANI     M229  ; 強制運轉模式
      ANI     M232  ; 自動模式KP
      OUT     M231  ; 手動步進訊號
281   LDI     M1672  ; 主傳動異常
      OR      SM400
      ANI     M1730  ; 出料空氣壓力異常
      OUT     M900  ; 強制運轉模式條件
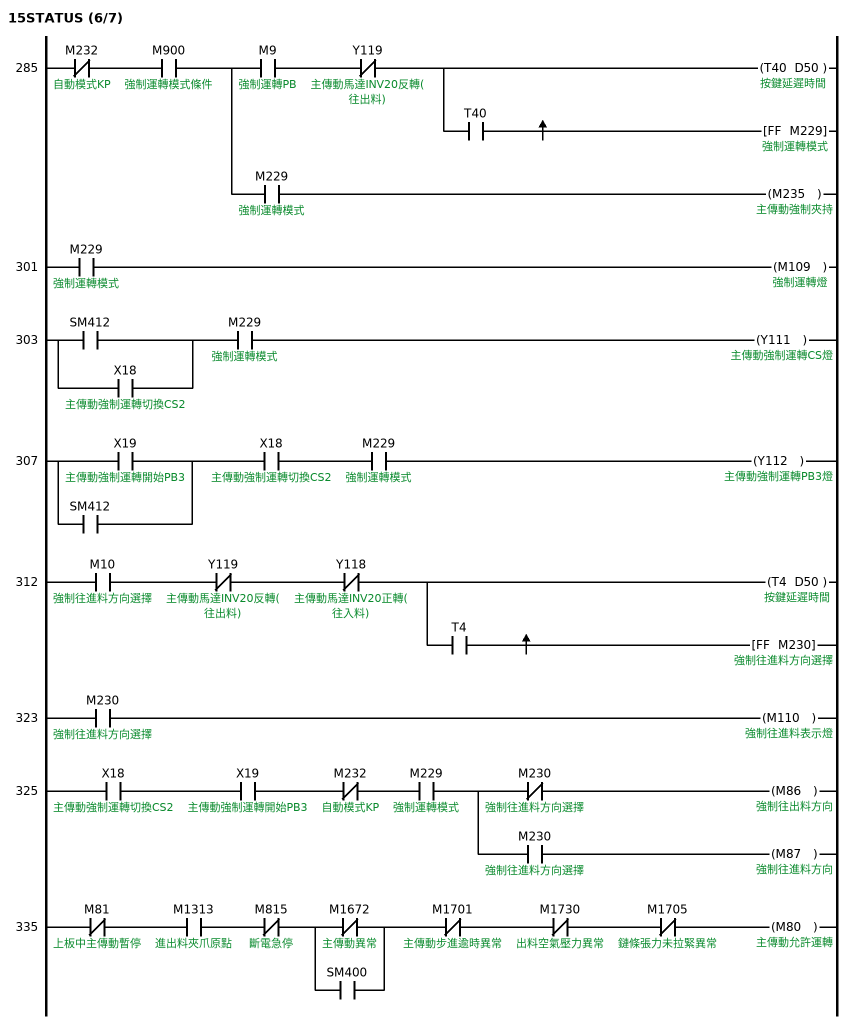
285   LDI     M232  ; 自動模式KP
      AND     M900  ; 強制運轉模式條件
      MPS
      AND     M9  ; 強制運轉PB
      ANI     Y119  ; 主傳動馬達INV20反轉(往出料)
      OUT     T40 D50  ; 按鍵延遲時間
      AND     T40
      MEP
      FF      M229
      MPP
      AND     M229  ; 強制運轉模式
      OUT     M235  ; 主傳動強制夾持
301   LD      M229  ; 強制運轉模式
      OUT     M109  ; 強制運轉燈
303   LD      SM412
      OR      X18  ; 主傳動強制運轉切換CS2
      AND     M229  ; 強制運轉模式
      OUT     Y111  ; 主傳動強制運轉CS燈
307   LD      X19  ; 主傳動強制運轉開始PB3
      OR      SM412
      AND     X18  ; 主傳動強制運轉切換CS2
      AND     M229  ; 強制運轉模式
      OUT     Y112  ; 主傳動強制運轉PB3燈
312   LD      M10  ; 強制往進料方向選擇
      ANI     Y119  ; 主傳動馬達INV20反轉(往出料)
      ANI     Y118  ; 主傳動馬達INV20正轉(往入料)
      OUT     T4 D50  ; 按鍵延遲時間
      AND     T4
      MEP
      FF      M230  ; 強制往進料方向選擇
323   LD      M230  ; 強制往進料方向選擇
      OUT     M110  ; 強制往進料表示燈
325   LD      X18  ; 主傳動強制運轉切換CS2
      AND     X19  ; 主傳動強制運轉開始PB3
      ANI     M232  ; 自動模式KP
      AND     M229  ; 強制運轉模式
      MPS
      ANI     M230  ; 強制往進料方向選擇
      OUT     M86  ; 強制往出料方向
      MPP
      AND     M230  ; 強制往進料方向選擇
      OUT     M87  ; 強制往進料方向
335   LDI     M81  ; 上板中主傳動暫停
      AND     M1313  ; 進出料夾爪原點
      ANI     M815  ; 斷電急停
      LDI     M1672  ; 主傳動異常
      OR      SM400
      ANB
      ANI     M1701  ; 主傳動步進逾時異常
      ANI     M1730  ; 出料空氣壓力異常
      ANI     M1705  ; 鏈條張力未拉緊異常
      OUT     M80  ; 主傳動允許運轉
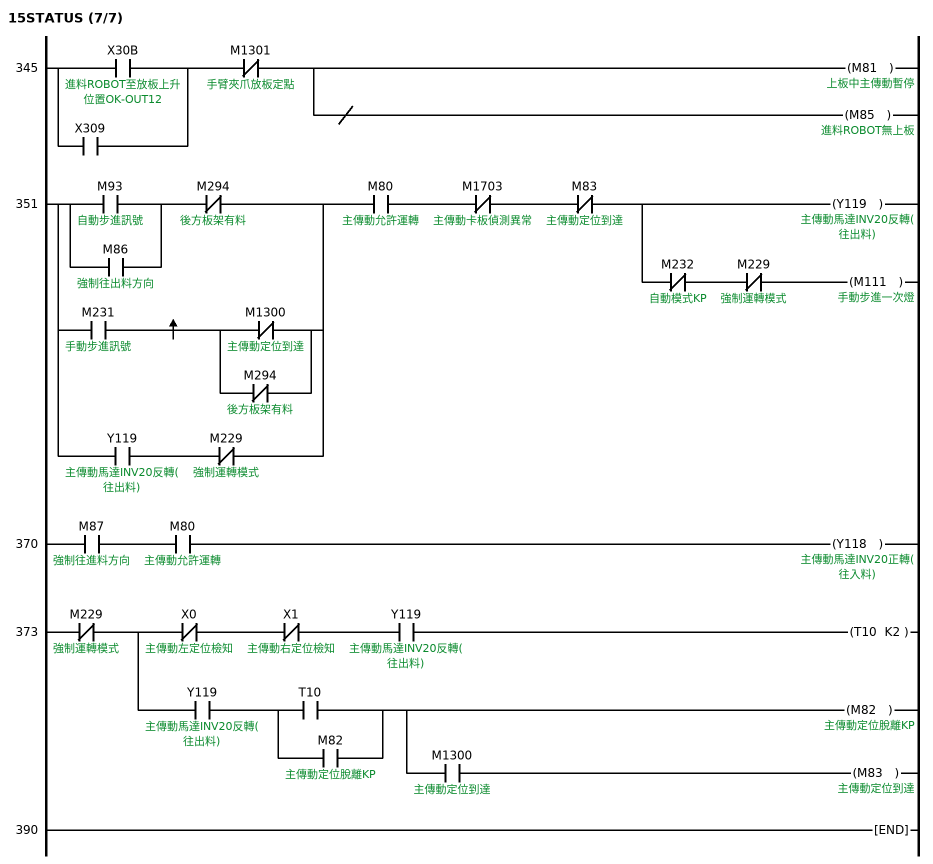
345   LD      X30B  ; 進料ROBOT至放板上升位置OK-OUT12
      OR      X309
      ANI     M1301  ; 手臂夾爪放板定點
      OUT     M81  ; 上板中主傳動暫停
      INV
      OUT     M85  ; 進料ROBOT無上板
351   LD      M93  ; 自動步進訊號
      OR      M86  ; 強制往出料方向
      ANI     M294  ; 後方板架有料
      LD      M231  ; 手動步進訊號
      MEP
      LDI     M1300  ; 主傳動定位到達
      ORI     M294  ; 後方板架有料
      ANB
      ORB
      LD      Y119  ; 主傳動馬達INV20反轉(往出料)
      ANI     M229  ; 強制運轉模式
      ORB
      AND     M80  ; 主傳動允許運轉
      ANI     M1703  ; 主傳動卡板偵測異常
      ANI     M83  ; 主傳動定位到達
      OUT     Y119  ; 主傳動馬達INV20反轉(往出料)
      ANI     M232  ; 自動模式KP
      ANI     M229  ; 強制運轉模式
      OUT     M111  ; 手動步進一次燈
370   LD      M87  ; 強制往進料方向
      AND     M80  ; 主傳動允許運轉
      OUT     Y118  ; 主傳動馬達INV20正轉(往入料)
373   LDI     M229  ; 強制運轉模式
      MPS
      ANI     X0  ; 主傳動左定位檢知
      ANI     X1  ; 主傳動右定位檢知
      AND     Y119  ; 主傳動馬達INV20反轉(往出料)
      OUT     T10 K2
      MPP
      AND     Y119  ; 主傳動馬達INV20反轉(往出料)
      LD      T10
      OR      M82  ; 主傳動定位脫離KP
      ANB
      OUT     M82  ; 主傳動定位脫離KP
      AND     M1300  ; 主傳動定位到達
      OUT     M83  ; 主傳動定位到達
390   END
END_PROGRAM

PROGRAM 16ETHERN
